LIN {X 0,Y 707.788,Z 622.318,A -85,B 0,C 180,E1 3542.213,E2 3542.213} C_VEL
LIN {X 0,Y 698.542,Z 601.31,A -85,B 0,C 180,E1 3542.971,E2 3542.971} C_VEL
LIN {X 0,Y 698.282,Z 601.31,A -85,B 0,C 180,E1 3548.645,E2 3548.645} C_VEL
LIN {X 0,Y 698.409,Z 601.31,A -85,B 0,C 180,E1 3554.29,E2 3554.29} C_VEL
LIN {X 0,Y 698.252,Z 601.31,A -85,B 0,C 180,E1 3559.425,E2 3559.425} C_VEL
LIN {X 0,Y 698.249,Z 601.31,A -85,B 0,C 180,E1 3564.14,E2 3564.14} C_VEL
LIN {X 0,Y 698.337,Z 601.31,A -85,B 0,C 180,E1 3568.624,E2 3568.624} C_VEL
LIN {X 0,Y 698.426,Z 601.31,A -85,B 0,C 180,E1 3572.902,E2 3572.902} C_VEL
LIN {X 0,Y 698.537,Z 601.31,A -85,B 0,C 180,E1 3577.022,E2 3577.022} C_VEL
LIN {X 0,Y 698.549,Z 601.31,A -85,B 0,C 180,E1 3582.641,E2 3582.641} C_VEL
LIN {X 0,Y 698.415,Z 601.31,A -85,B 0,C 180,E1 3587.509,E2 3587.509} C_VEL
LIN {X 0,Y 698.636,Z 601.31,A -85,B 0,C 180,E1 3592.523,E2 3592.523} C_VEL
LIN {X 0,Y 698.754,Z 601.31,A -85,B 0,C 180,E1 3597.513,E2 3597.513} C_VEL
LIN {X 0,Y 698.624,Z 601.31,A -85,B 0,C 180,E1 3602.484,E2 3602.484} C_VEL
LIN {X 0,Y 698.589,Z 601.31,A -85,B 0,C 180,E1 3606.223,E2 3606.223} C_VEL
LIN {X 0,Y 698.52,Z 601.31,A -85,B 0,C 180,E1 3611.254,E2 3611.254} C_VEL
LIN {X 0,Y 698.581,Z 601.31,A -85,B 0,C 180,E1 3616.372,E2 3616.372} C_VEL
LIN {X 0,Y 698.492,Z 601.31,A -85,B 0,C 180,E1 3621.633,E2 3621.633} C_VEL
LIN {X 0,Y 698.439,Z 601.31,A -85,B 0,C 180,E1 3625.707,E2 3625.707} C_VEL
LIN {X 0,Y 698.346,Z 601.31,A -85,B 0,C 180,E1 3629.927,E2 3629.927} C_VEL
LIN {X 0,Y 698.291,Z 601.31,A -85,B 0,C 180,E1 3634.451,E2 3634.451} C_VEL
LIN {X 0,Y 698.292,Z 601.31,A -85,B 0,C 180,E1 3638.984,E2 3638.984} C_VEL
LIN {X 0,Y 698.437,Z 601.31,A -85,B 0,C 180,E1 3644.277,E2 3644.277} C_VEL
LIN {X 0,Y 698.295,Z 601.31,A -85,B 0,C 180,E1 3649.399,E2 3649.399} C_VEL
LIN {X 0,Y 698.256,Z 601.31,A -85,B 0,C 180,E1 3654.13,E2 3654.13} C_VEL
LIN {X 0,Y 698.361,Z 601.31,A -85,B 0,C 180,E1 3658.616,E2 3658.616} C_VEL
LIN {X 0,Y 698.567,Z 601.31,A -85,B 0,C 180,E1 3664.287,E2 3664.287} C_VEL
LIN {X 0,Y 698.644,Z 601.31,A -85,B 0,C 180,E1 3665.087,E2 3665.087} C_VEL
LIN {X 0,Y 704.33,Z 620.623,A -85,B 0,C 180,E1 3665.608,E2 3665.608} C_VEL
LIN {X 0,Y 703.741,Z 661.307,A -85,B 0,C 180,E1 3666.603,E2 3666.603} C_VEL
LIN {X 0,Y 702.767,Z 699.55,A -85,B 0,C 180,E1 3668.056,E2 3668.056} C_VEL
LIN {X 0,Y 701.625,Z 735.549,A -85,B 0,C 180,E1 3669.988,E2 3669.988} C_VEL
LIN {X 0,Y 700.652,Z 767.288,A -85,B 0,C 180,E1 3672.261,E2 3672.261} C_VEL
LIN {X 0,Y 699.841,Z 795.512,A -85,B 0,C 180,E1 3674.938,E2 3674.938} C_VEL
LIN {X 0,Y 699.357,Z 818.283,A -85,B 0,C 180,E1 3677.801,E2 3677.801} C_VEL
LIN {X 0,Y 699.049,Z 835.787,A -85,B 0,C 180,E1 3680.796,E2 3680.796} C_VEL
LIN {X 0,Y 698.89,Z 847.743,A -85,B 0,C 180,E1 3683.773,E2 3683.773} C_VEL
LIN {X 0,Y 698.874,Z 854.031,A -85,B 0,C 180,E1 3686.267,E2 3686.267} C_VEL
LIN {X 0,Y 698.804,Z 857.085,A -85,B 0,C 180,E1 3688.754,E2 3688.754} C_VEL
LIN {X 0,Y 698.887,Z 857.026,A -85,B 0,C 180,E1 3691.239,E2 3691.239} C_VEL
LIN {X 0,Y 698.999,Z 852.206,A -85,B 0,C 180,E1 3694.519,E2 3694.519} C_VEL
LIN {X 0,Y 699.071,Z 841.77,A -85,B 0,C 180,E1 3697.782,E2 3697.782} C_VEL
LIN {X 0,Y 699.25,Z 825.88,A -85,B 0,C 180,E1 3700.926,E2 3700.926} C_VEL
LIN {X 0,Y 699.701,Z 804.549,A -85,B 0,C 180,E1 3703.937,E2 3703.937} C_VEL
LIN {X 0,Y 700.362,Z 778.69,A -85,B 0,C 180,E1 3706.654,E2 3706.654} C_VEL
LIN {X 0,Y 701.32,Z 747.571,A -85,B 0,C 180,E1 3709.129,E2 3709.129} C_VEL
LIN {X 0,Y 702.354,Z 713.484,A -85,B 0,C 180,E1 3711.18,E2 3711.18} C_VEL
LIN {X 0,Y 703.382,Z 676.025,A -85,B 0,C 180,E1 3712.811,E2 3712.811} C_VEL
LIN {X 0,Y 704.233,Z 635.503,A -85,B 0,C 180,E1 3714,E2 3714} C_VEL
LIN {X 0,Y 703.617,Z 616.54,A -85,B 0,C 180,E1 3714.405,E2 3714.405} C_VEL
LIN {X 0,Y 698.364,Z 601.31,A -85,B 0,C 180,E1 3714.86,E2 3714.86} C_VEL
LIN {X 0,Y 698.363,Z 601.31,A -85,B 0,C 180,E1 3719.931,E2 3719.931} C_VEL
LIN {X 0,Y 698.307,Z 601.31,A -85,B 0,C 180,E1 3724.479,E2 3724.479} C_VEL
LIN {X 0,Y 698.251,Z 601.31,A -85,B 0,C 180,E1 3728.994,E2 3728.994} C_VEL
LIN {X 0,Y 698.44,Z 601.31,A -85,B 0,C 180,E1 3734.297,E2 3734.297} C_VEL
LIN {X 0,Y 698.27,Z 601.31,A -85,B 0,C 180,E1 3739.413,E2 3739.413} C_VEL
LIN {X 0,Y 698.252,Z 601.31,A -85,B 0,C 180,E1 3744.144,E2 3744.144} C_VEL
LIN {X 0,Y 698.338,Z 601.31,A -85,B 0,C 180,E1 3748.628,E2 3748.628} C_VEL
LIN {X 0,Y 698.504,Z 601.31,A -85,B 0,C 180,E1 3754.296,E2 3754.296} C_VEL
LIN {X 0,Y 698.327,Z 601.31,A -85,B 0,C 180,E1 3758.897,E2 3758.897} C_VEL
LIN {X 0,Y 698.394,Z 601.31,A -85,B 0,C 180,E1 3761.57,E2 3761.57} C_VEL
LIN {X 0,Y 702.105,Z 618.347,A -85,B 0,C 180,E1 3761.867,E2 3761.867} C_VEL
LIN {X 0,Y 701.839,Z 691.618,A -85,B 0,C 180,E1 3762.737,E2 3762.737} C_VEL
LIN {X 0,Y 701.426,Z 724.721,A -85,B 0,C 180,E1 3763.615,E2 3763.615} C_VEL
LIN {X 0,Y 700.738,Z 756.316,A -85,B 0,C 180,E1 3764.966,E2 3764.966} C_VEL
LIN {X 0,Y 700.111,Z 785.157,A -85,B 0,C 180,E1 3766.752,E2 3766.752} C_VEL
LIN {X 0,Y 699.572,Z 810.159,A -85,B 0,C 180,E1 3768.921,E2 3768.921} C_VEL
LIN {X 0,Y 699.205,Z 830.58,A -85,B 0,C 180,E1 3771.435,E2 3771.435} C_VEL
LIN {X 0,Y 699.029,Z 845.13,A -85,B 0,C 180,E1 3774.093,E2 3774.093} C_VEL
LIN {X 0,Y 698.976,Z 854.196,A -85,B 0,C 180,E1 3776.896,E2 3776.896} C_VEL
LIN {X 0,Y 698.914,Z 856.955,A -85,B 0,C 180,E1 3778.76,E2 3778.76} C_VEL
LIN {X 0,Y 698.933,Z 856.877,A -85,B 0,C 180,E1 3781.244,E2 3781.244} C_VEL
LIN {X 0,Y 699.024,Z 851.303,A -85,B 0,C 180,E1 3784.126,E2 3784.126} C_VEL
LIN {X 0,Y 699.113,Z 840.282,A -85,B 0,C 180,E1 3786.846,E2 3786.846} C_VEL
LIN {X 0,Y 699.33,Z 823.303,A -85,B 0,C 180,E1 3789.477,E2 3789.477} C_VEL
LIN {X 0,Y 699.742,Z 800.952,A -85,B 0,C 180,E1 3791.87,E2 3791.87} C_VEL
LIN {X 0,Y 700.299,Z 777.418,A -85,B 0,C 180,E1 3793.701,E2 3793.701} C_VEL
LIN {X 0,Y 696.623,Z 764.377,A -85,B 0,C 180,E1 3794.621,E2 3794.621} C_VEL
LIN {X 0,Y 693.254,Z 752.31,A -85,B 0,C 180,E1 3795.348,E2 3795.348} C_VEL
LIN {X 0,Y 693.225,Z 750.405,A -85,B 0,C 180,E1 3795.44,E2 3795.44} C_VEL
LIN {X 0,Y 693.951,Z 717.579,A -85,B 0,C 180,E1 3796.733,E2 3796.733} C_VEL
LIN {X 0,Y 694.411,Z 682.542,A -85,B 0,C 180,E1 3797.539,E2 3797.539} C_VEL
LIN {X 0,Y 694.009,Z 612.919,A -85,B 0,C 180,E1 3798.371,E2 3798.371} C_VEL
LIN {X 0,Y 690.712,Z 601.31,A -85,B 0,C 180,E1 3798.635,E2 3798.635} C_VEL
LIN {X 0,Y 690.49,Z 601.31,A -85,B 0,C 180,E1 3803.262,E2 3803.262} C_VEL
LIN {X 0,Y 690.484,Z 601.31,A -85,B 0,C 180,E1 3808.634,E2 3808.634} C_VEL
LIN {X 0,Y 690.388,Z 601.31,A -85,B 0,C 180,E1 3813.495,E2 3813.495} C_VEL
LIN {X 0,Y 690.456,Z 601.31,A -85,B 0,C 180,E1 3817.905,E2 3817.905} C_VEL
LIN {X 0,Y 690.503,Z 601.31,A -85,B 0,C 180,E1 3823.608,E2 3823.608} C_VEL
LIN {X 0,Y 690.271,Z 601.31,A -85,B 0,C 180,E1 3828.817,E2 3828.817} C_VEL
LIN {X 0,Y 690.311,Z 601.31,A -85,B 0,C 180,E1 3833.66,E2 3833.66} C_VEL
LIN {X 0,Y 690.363,Z 602.018,A -85,B 0,C 180,E1 3836.624,E2 3836.624} C_VEL
LIN {X 0,Y 701.618,Z 627.968,A -85,B 0,C 180,E1 3837.536,E2 3837.536} C_VEL
LIN {X 0,Y 701.063,Z 707.913,A -85,B 0,C 180,E1 3838.565,E2 3838.565} C_VEL
LIN {X 0,Y 700.009,Z 748.6,A -85,B 0,C 180,E1 3839.519,E2 3839.519} C_VEL
LIN {X 0,Y 698.553,Z 792.111,A -85,B 0,C 180,E1 3841.059,E2 3841.059} C_VEL
LIN {X 0,Y 696.858,Z 832.632,A -85,B 0,C 180,E1 3843.039,E2 3843.039} C_VEL
LIN {X 0,Y 695.161,Z 870.148,A -85,B 0,C 180,E1 3845.431,E2 3845.431} C_VEL
LIN {X 0,Y 693.739,Z 904.255,A -85,B 0,C 180,E1 3848.208,E2 3848.208} C_VEL
LIN {X 0,Y 692.563,Z 934.568,A -85,B 0,C 180,E1 3851.343,E2 3851.343} C_VEL
LIN {X 0,Y 691.764,Z 961.239,A -85,B 0,C 180,E1 3854.927,E2 3854.927} C_VEL
LIN {X 0,Y 691.258,Z 981.632,A -85,B 0,C 180,E1 3858.626,E2 3858.626} C_VEL
LIN {X 0,Y 691.102,Z 994.244,A -85,B 0,C 180,E1 3861.81,E2 3861.81} C_VEL
LIN {X 0,Y 690.958,Z 1003.715,A -85,B 0,C 180,E1 3865.625,E2 3865.625} C_VEL
LIN {X 0,Y 691.006,Z 1007.169,A -85,B 0,C 180,E1 3868.747,E2 3868.747} C_VEL
LIN {X 0,Y 691.033,Z 1006.216,A -85,B 0,C 180,E1 3872.517,E2 3872.517} C_VEL
LIN {X 0,Y 690.976,Z 999.627,A -85,B 0,C 180,E1 3876.298,E2 3876.298} C_VEL
LIN {X 0,Y 691.137,Z 988.788,A -85,B 0,C 180,E1 3879.717,E2 3879.717} C_VEL
LIN {X 0,Y 691.37,Z 970.858,A -85,B 0,C 180,E1 3883.475,E2 3883.475} C_VEL
LIN {X 0,Y 691.911,Z 949.955,A -85,B 0,C 180,E1 3886.707,E2 3886.707} C_VEL
LIN {X 0,Y 692.876,Z 923.253,A -85,B 0,C 180,E1 3889.921,E2 3889.921} C_VEL
LIN {X 0,Y 694.331,Z 889.898,A -85,B 0,C 180,E1 3893.048,E2 3893.048} C_VEL
LIN {X 0,Y 696.009,Z 851.914,A -85,B 0,C 180,E1 3895.814,E2 3895.814} C_VEL
LIN {X 0,Y 697.776,Z 811.008,A -85,B 0,C 180,E1 3898.09,E2 3898.09} C_VEL
LIN {X 0,Y 699.268,Z 772.005,A -85,B 0,C 180,E1 3899.718,E2 3899.718} C_VEL
LIN {X 0,Y 700.658,Z 729.711,A -85,B 0,C 180,E1 3900.979,E2 3900.979} C_VEL
LIN {X 0,Y 701.336,Z 686.179,A -85,B 0,C 180,E1 3901.776,E2 3901.776} C_VEL
LIN {X 0,Y 701.268,Z 625.08,A -85,B 0,C 180,E1 3902.516,E2 3902.516} C_VEL
LIN {X 0,Y 690.525,Z 601.31,A -85,B 0,C 180,E1 3903.414,E2 3903.414} C_VEL
LIN {X 0,Y 690.391,Z 601.31,A -85,B 0,C 180,E1 3907.921,E2 3907.921} C_VEL
LIN {X 0,Y 690.469,Z 601.31,A -85,B 0,C 180,E1 3913.611,E2 3913.611} C_VEL
LIN {X 0,Y 690.275,Z 601.31,A -85,B 0,C 180,E1 3918.821,E2 3918.821} C_VEL
LIN {X 0,Y 690.342,Z 601.31,A -85,B 0,C 180,E1 3923.664,E2 3923.664} C_VEL
LIN {X 0,Y 690.429,Z 601.31,A -85,B 0,C 180,E1 3928.865,E2 3928.865} C_VEL
LIN {X 0,Y 690.568,Z 601.31,A -85,B 0,C 180,E1 3934.113,E2 3934.113} C_VEL
LIN {X 0,Y 690.562,Z 601.31,A -85,B 0,C 180,E1 3938.102,E2 3938.102} C_VEL
LIN {X 0,Y 690.617,Z 601.31,A -85,B 0,C 180,E1 3943.43,E2 3943.43} C_VEL
LIN {X 0,Y 690.638,Z 601.31,A -85,B 0,C 180,E1 3948.613,E2 3948.613} C_VEL
LIN {X 0,Y 690.785,Z 601.31,A -85,B 0,C 180,E1 3953.703,E2 3953.703} C_VEL
LIN {X 0,Y 690.738,Z 601.31,A -85,B 0,C 180,E1 3958.742,E2 3958.742} C_VEL
LIN {X 0,Y 690.741,Z 601.31,A -85,B 0,C 180,E1 3962.512,E2 3962.512} C_VEL
LIN {X 0,Y 690.68,Z 601.31,A -85,B 0,C 180,E1 3966.294,E2 3966.294} C_VEL
LIN {X 0,Y 690.644,Z 601.31,A -85,B 0,C 180,E1 3971.384,E2 3971.384} C_VEL
LIN {X 0,Y 690.683,Z 601.31,A -85,B 0,C 180,E1 3976.565,E2 3976.565} C_VEL
LIN {X 0,Y 690.558,Z 601.31,A -85,B 0,C 180,E1 3981.895,E2 3981.895} C_VEL
LIN {X 0,Y 690.505,Z 601.31,A -85,B 0,C 180,E1 3986.024,E2 3986.024} C_VEL
LIN {X 0,Y 690.432,Z 601.31,A -85,B 0,C 180,E1 3991.136,E2 3991.136} C_VEL
LIN {X 0,Y 690.429,Z 601.31,A -85,B 0,C 180,E1 3996.326,E2 3996.326} C_VEL
LIN {X 0,Y 690.409,Z 601.31,A -85,B 0,C 180,E1 4001.734,E2 4001.734} C_VEL
LIN {X 0,Y 690.35,Z 601.31,A -85,B 0,C 180,E1 4006.395,E2 4006.395} C_VEL
LIN {X 0,Y 690.377,Z 601.31,A -85,B 0,C 180,E1 4012.177,E2 4012.177} C_VEL
LIN {X 0,Y 690.34,Z 601.31,A -85,B 0,C 180,E1 4016.717,E2 4016.717} C_VEL
LIN {X 0,Y 690.493,Z 601.31,A -85,B 0,C 180,E1 4021.347,E2 4021.347} C_VEL
LIN {X 0,Y 690.725,Z 601.31,A -85,B 0,C 180,E1 4024.781,E2 4024.781} C_VEL
LIN {X 0,Y 697.118,Z 622.821,A -85,B 0,C 180,E1 4025.383,E2 4025.383} C_VEL
LIN {X 0,Y 696.426,Z 663.052,A -85,B 0,C 180,E1 4026.397,E2 4026.397} C_VEL
LIN {X 0,Y 695.307,Z 700.604,A -85,B 0,C 180,E1 4027.861,E2 4027.861} C_VEL
LIN {X 0,Y 694.055,Z 736.725,A -85,B 0,C 180,E1 4029.836,E2 4029.836} C_VEL
LIN {X 0,Y 692.938,Z 768.609,A -85,B 0,C 180,E1 4032.17,E2 4032.17} C_VEL
LIN {X 0,Y 692.103,Z 795.501,A -85,B 0,C 180,E1 4034.765,E2 4034.765} C_VEL
LIN {X 0,Y 691.527,Z 818.279,A -85,B 0,C 180,E1 4037.661,E2 4037.661} C_VEL
LIN {X 0,Y 691.197,Z 834.771,A -85,B 0,C 180,E1 4040.48,E2 4040.48} C_VEL
LIN {X 0,Y 690.996,Z 847.743,A -85,B 0,C 180,E1 4043.702,E2 4043.702} C_VEL
LIN {X 0,Y 690.984,Z 854.033,A -85,B 0,C 180,E1 4046.225,E2 4046.225} C_VEL
LIN {X 0,Y 690.911,Z 857.08,A -85,B 0,C 180,E1 4048.74,E2 4048.74} C_VEL
LIN {X 0,Y 690.989,Z 857.021,A -85,B 0,C 180,E1 4051.253,E2 4051.253} C_VEL
LIN {X 0,Y 691.099,Z 852.201,A -85,B 0,C 180,E1 4054.571,E2 4054.571} C_VEL
LIN {X 0,Y 691.166,Z 841.774,A -85,B 0,C 180,E1 4057.872,E2 4057.872} C_VEL
LIN {X 0,Y 691.426,Z 825.878,A -85,B 0,C 180,E1 4061.051,E2 4061.051} C_VEL
LIN {X 0,Y 691.895,Z 804.554,A -85,B 0,C 180,E1 4064.097,E2 4064.097} C_VEL
LIN {X 0,Y 692.653,Z 778.7,A -85,B 0,C 180,E1 4066.845,E2 4066.845} C_VEL
LIN {X 0,Y 693.687,Z 748.784,A -85,B 0,C 180,E1 4069.261,E2 4069.261} C_VEL
LIN {X 0,Y 694.853,Z 715.017,A -85,B 0,C 180,E1 4071.336,E2 4071.336} C_VEL
LIN {X 0,Y 695.978,Z 678.621,A -85,B 0,C 180,E1 4072.972,E2 4072.972} C_VEL
LIN {X 0,Y 696.933,Z 637.993,A -85,B 0,C 180,E1 4074.205,E2 4074.205} C_VEL
LIN {X 0,Y 696.408,Z 618.768,A -85,B 0,C 180,E1 4074.632,E2 4074.632} C_VEL
LIN {X 0,Y 690.439,Z 601.31,A -85,B 0,C 180,E1 4075.145,E2 4075.145} C_VEL
LIN {X 0,Y 690.421,Z 601.31,A -85,B 0,C 180,E1 4080.311,E2 4080.311} C_VEL
LIN {X 0,Y 690.396,Z 601.31,A -85,B 0,C 180,E1 4085.725,E2 4085.725} C_VEL
LIN {X 0,Y 690.327,Z 601.31,A -85,B 0,C 180,E1 4091.179,E2 4091.179} C_VEL
LIN {X 0,Y 690.433,Z 601.31,A -85,B 0,C 180,E1 4095.405,E2 4095.405} C_VEL
LIN {X 0,Y 690.317,Z 601.31,A -85,B 0,C 180,E1 4100.478,E2 4100.478} C_VEL
LIN {X 0,Y 690.325,Z 601.31,A -85,B 0,C 180,E1 4105.213,E2 4105.213} C_VEL
LIN {X 0,Y 690.402,Z 601.31,A -85,B 0,C 180,E1 4109.693,E2 4109.693} C_VEL
LIN {X 0,Y 690.587,Z 601.31,A -85,B 0,C 180,E1 4114.094,E2 4114.094} C_VEL
LIN {X 0,Y 690.488,Z 601.31,A -85,B 0,C 180,E1 4118.103,E2 4118.103} C_VEL
LIN {X 0,Y 690.45,Z 601.31,A -85,B 0,C 180,E1 4121.341,E2 4121.341} C_VEL
LIN {X 0,Y 694.653,Z 618.658,A -85,B 0,C 180,E1 4121.655,E2 4121.655} C_VEL
LIN {X 0,Y 694.336,Z 690.008,A -85,B 0,C 180,E1 4122.504,E2 4122.504} C_VEL
LIN {X 0,Y 693.867,Z 723.802,A -85,B 0,C 180,E1 4123.391,E2 4123.391} C_VEL
LIN {X 0,Y 693.115,Z 754.803,A -85,B 0,C 180,E1 4124.699,E2 4124.699} C_VEL
LIN {X 0,Y 692.445,Z 783.749,A -85,B 0,C 180,E1 4126.482,E2 4126.482} C_VEL
LIN {X 0,Y 691.778,Z 808.559,A -85,B 0,C 180,E1 4128.635,E2 4128.635} C_VEL
LIN {X 0,Y 691.41,Z 828.174,A -85,B 0,C 180,E1 4130.987,E2 4130.987} C_VEL
LIN {X 0,Y 691.181,Z 843.788,A -85,B 0,C 180,E1 4133.71,E2 4133.71} C_VEL
LIN {X 0,Y 691.113,Z 852.678,A -85,B 0,C 180,E1 4136.231,E2 4136.231} C_VEL
LIN {X 0,Y 691.021,Z 856.954,A -85,B 0,C 180,E1 4138.745,E2 4138.745} C_VEL
LIN {X 0,Y 691.038,Z 856.877,A -85,B 0,C 180,E1 4141.258,E2 4141.258} C_VEL
LIN {X 0,Y 691.125,Z 851.49,A -85,B 0,C 180,E1 4144.112,E2 4144.112} C_VEL
LIN {X 0,Y 691.229,Z 840.285,A -85,B 0,C 180,E1 4146.925,E2 4146.925} C_VEL
LIN {X 0,Y 691.469,Z 823.248,A -85,B 0,C 180,E1 4149.593,E2 4149.593} C_VEL
LIN {X 0,Y 691.942,Z 800.972,A -85,B 0,C 180,E1 4152.006,E2 4152.006} C_VEL
LIN {X 0,Y 692.635,Z 775.636,A -85,B 0,C 180,E1 4154.003,E2 4154.003} C_VEL
LIN {X 0,Y 693.225,Z 750.405,A -85,B 0,C 180,E1 4155.44,E2 4155.44} C_VEL
LIN {X 0,Y 689.935,Z 735.712,A -85,B 0,C 180,E1 4156.19,E2 4156.19} C_VEL
LIN {X 0,Y 686.319,Z 721.512,A -85,B 0,C 180,E1 4156.808,E2 4156.808} C_VEL
LIN {X 0,Y 686.329,Z 720.499,A -85,B 0,C 180,E1 4156.843,E2 4156.843} C_VEL
LIN {X 0,Y 686.892,Z 685.627,A -85,B 0,C 180,E1 4157.696,E2 4157.696} C_VEL
LIN {X 0,Y 686.499,Z 613.882,A -85,B 0,C 180,E1 4158.596,E2 4158.596} C_VEL
LIN {X 0,Y 682.779,Z 601.31,A -85,B 0,C 180,E1 4158.92,E2 4158.92} C_VEL
LIN {X 0,Y 682.567,Z 601.31,A -85,B 0,C 180,E1 4164.483,E2 4164.483} C_VEL
LIN {X 0,Y 682.51,Z 601.31,A -85,B 0,C 180,E1 4169.231,E2 4169.231} C_VEL
LIN {X 0,Y 682.523,Z 601.31,A -85,B 0,C 180,E1 4174.781,E2 4174.781} C_VEL
LIN {X 0,Y 682.402,Z 601.31,A -85,B 0,C 180,E1 4180.076,E2 4180.076} C_VEL
LIN {X 0,Y 682.593,Z 601.31,A -85,B 0,C 180,E1 4184.743,E2 4184.743} C_VEL
LIN {X 0,Y 682.366,Z 601.31,A -85,B 0,C 180,E1 4189.918,E2 4189.918} C_VEL
LIN {X 0,Y 682.375,Z 601.31,A -85,B 0,C 180,E1 4195.228,E2 4195.228} C_VEL
LIN {X 0,Y 682.39,Z 601.31,A -85,B 0,C 180,E1 4196.166,E2 4196.166} C_VEL
LIN {X 0,Y 694.974,Z 629.987,A -85,B 0,C 180,E1 4197.212,E2 4197.212} C_VEL
LIN {X 0,Y 694.299,Z 708.221,A -85,B 0,C 180,E1 4198.229,E2 4198.229} C_VEL
LIN {X 0,Y 693.162,Z 748.575,A -85,B 0,C 180,E1 4199.185,E2 4199.185} C_VEL
LIN {X 0,Y 691.58,Z 791.241,A -85,B 0,C 180,E1 4200.702,E2 4200.702} C_VEL
LIN {X 0,Y 689.771,Z 830.846,A -85,B 0,C 180,E1 4202.636,E2 4202.636} C_VEL
LIN {X 0,Y 687.947,Z 867.704,A -85,B 0,C 180,E1 4204.972,E2 4204.972} C_VEL
LIN {X 0,Y 686.216,Z 902.493,A -85,B 0,C 180,E1 4207.786,E2 4207.786} C_VEL
LIN {X 0,Y 684.879,Z 934.568,A -85,B 0,C 180,E1 4211.125,E2 4211.125} C_VEL
LIN {X 0,Y 683.955,Z 961.237,A -85,B 0,C 180,E1 4214.751,E2 4214.751} C_VEL
LIN {X 0,Y 683.396,Z 981.631,A -85,B 0,C 180,E1 4218.493,E2 4218.493} C_VEL
LIN {X 0,Y 683.232,Z 994.244,A -85,B 0,C 180,E1 4221.715,E2 4221.715} C_VEL
LIN {X 0,Y 683.077,Z 1003.671,A -85,B 0,C 180,E1 4225.551,E2 4225.551} C_VEL
LIN {X 0,Y 683.103,Z 1007.169,A -85,B 0,C 180,E1 4228.733,E2 4228.733} C_VEL
LIN {X 0,Y 683.127,Z 1006.215,A -85,B 0,C 180,E1 4232.546,E2 4232.546} C_VEL
LIN {X 0,Y 683.155,Z 1001.188,A -85,B 0,C 180,E1 4235.732,E2 4235.732} C_VEL
LIN {X 0,Y 683.235,Z 989.724,A -85,B 0,C 180,E1 4239.572,E2 4239.572} C_VEL
LIN {X 0,Y 683.523,Z 973.523,A -85,B 0,C 180,E1 4243.137,E2 4243.137} C_VEL
LIN {X 0,Y 684.066,Z 952.358,A -85,B 0,C 180,E1 4246.573,E2 4246.573} C_VEL
LIN {X 0,Y 685.197,Z 924.381,A -85,B 0,C 180,E1 4250.034,E2 4250.034} C_VEL
LIN {X 0,Y 686.821,Z 889.899,A -85,B 0,C 180,E1 4253.315,E2 4253.315} C_VEL
LIN {X 0,Y 688.737,Z 851.914,A -85,B 0,C 180,E1 4256.107,E2 4256.107} C_VEL
LIN {X 0,Y 690.658,Z 810.743,A -85,B 0,C 180,E1 4258.419,E2 4258.419} C_VEL
LIN {X 0,Y 692.377,Z 770.375,A -85,B 0,C 180,E1 4260.105,E2 4260.105} C_VEL
LIN {X 0,Y 693.839,Z 729.451,A -85,B 0,C 180,E1 4261.324,E2 4261.324} C_VEL
LIN {X 0,Y 694.646,Z 685.297,A -85,B 0,C 180,E1 4262.131,E2 4262.131} C_VEL
LIN {X 0,Y 694.462,Z 627.246,A -85,B 0,C 180,E1 4262.849,E2 4262.849} C_VEL
LIN {X 0,Y 682.565,Z 601.31,A -85,B 0,C 180,E1 4263.847,E2 4263.847} C_VEL
LIN {X 0,Y 682.38,Z 601.31,A -85,B 0,C 180,E1 4269.011,E2 4269.011} C_VEL
LIN {X 0,Y 682.563,Z 601.31,A -85,B 0,C 180,E1 4273.49,E2 4273.49} C_VEL
LIN {X 0,Y 682.376,Z 601.31,A -85,B 0,C 180,E1 4279.028,E2 4279.028} C_VEL
LIN {X 0,Y 682.394,Z 601.31,A -85,B 0,C 180,E1 4283.172,E2 4283.172} C_VEL
LIN {X 0,Y 682.435,Z 601.31,A -85,B 0,C 180,E1 4287.806,E2 4287.806} C_VEL
LIN {X 0,Y 682.624,Z 601.31,A -85,B 0,C 180,E1 4292.614,E2 4292.614} C_VEL
LIN {X 0,Y 682.664,Z 601.31,A -85,B 0,C 180,E1 4297.835,E2 4297.835} C_VEL
LIN {X 0,Y 682.692,Z 601.31,A -85,B 0,C 180,E1 4303.232,E2 4303.232} C_VEL
LIN {X 0,Y 682.708,Z 601.31,A -85,B 0,C 180,E1 4308.479,E2 4308.479} C_VEL
LIN {X 0,Y 682.901,Z 601.31,A -85,B 0,C 180,E1 4313.63,E2 4313.63} C_VEL
LIN {X 0,Y 682.839,Z 601.31,A -85,B 0,C 180,E1 4318.727,E2 4318.727} C_VEL
LIN {X 0,Y 682.862,Z 601.31,A -85,B 0,C 180,E1 4323.068,E2 4323.068} C_VEL
LIN {X 0,Y 682.782,Z 601.31,A -85,B 0,C 180,E1 4327.648,E2 4327.648} C_VEL
LIN {X 0,Y 682.778,Z 601.31,A -85,B 0,C 180,E1 4332.817,E2 4332.817} C_VEL
LIN {X 0,Y 682.708,Z 601.31,A -85,B 0,C 180,E1 4338.097,E2 4338.097} C_VEL
LIN {X 0,Y 682.613,Z 601.31,A -85,B 0,C 180,E1 4343.543,E2 4343.543} C_VEL
LIN {X 0,Y 682.576,Z 601.31,A -85,B 0,C 180,E1 4347.777,E2 4347.777} C_VEL
LIN {X 0,Y 682.459,Z 601.31,A -85,B 0,C 180,E1 4352.463,E2 4352.463} C_VEL
LIN {X 0,Y 682.483,Z 601.31,A -85,B 0,C 180,E1 4356.936,E2 4356.936} C_VEL
LIN {X 0,Y 682.589,Z 601.31,A -85,B 0,C 180,E1 4362.896,E2 4362.896} C_VEL
LIN {X 0,Y 682.407,Z 601.31,A -85,B 0,C 180,E1 4368.227,E2 4368.227} C_VEL
LIN {X 0,Y 682.408,Z 601.31,A -85,B 0,C 180,E1 4373.161,E2 4373.161} C_VEL
LIN {X 0,Y 682.467,Z 601.31,A -85,B 0,C 180,E1 4377.798,E2 4377.798} C_VEL
LIN {X 0,Y 682.663,Z 601.31,A -85,B 0,C 180,E1 4382.574,E2 4382.574} C_VEL
LIN {X 0,Y 682.799,Z 601.31,A -85,B 0,C 180,E1 4384.457,E2 4384.457} C_VEL
LIN {X 0,Y 689.909,Z 624.36,A -85,B 0,C 180,E1 4385.14,E2 4385.14} C_VEL
LIN {X 0,Y 689.131,Z 663.874,A -85,B 0,C 180,E1 4386.158,E2 4386.158} C_VEL
LIN {X 0,Y 687.857,Z 701.615,A -85,B 0,C 180,E1 4387.66,E2 4387.66} C_VEL
LIN {X 0,Y 686.463,Z 738.394,A -85,B 0,C 180,E1 4389.713,E2 4389.713} C_VEL
LIN {X 0,Y 685.205,Z 770.515,A -85,B 0,C 180,E1 4392.129,E2 4392.129} C_VEL
LIN {X 0,Y 684.235,Z 798.363,A -85,B 0,C 180,E1 4394.915,E2 4394.915} C_VEL
LIN {X 0,Y 683.661,Z 821.506,A -85,B 0,C 180,E1 4398.004,E2 4398.004} C_VEL
LIN {X 0,Y 683.26,Z 838.009,A -85,B 0,C 180,E1 4401.066,E2 4401.066} C_VEL
LIN {X 0,Y 683.161,Z 849.602,A -85,B 0,C 180,E1 4404.268,E2 4404.268} C_VEL
LIN {X 0,Y 683.114,Z 855.945,A -85,B 0,C 180,E1 4407.454,E2 4407.454} C_VEL
LIN {X 0,Y 683.008,Z 857.439,A -85,B 0,C 180,E1 4409.996,E2 4409.996} C_VEL
LIN {X 0,Y 683.084,Z 855.835,A -85,B 0,C 180,E1 4412.539,E2 4412.539} C_VEL
LIN {X 0,Y 683.172,Z 849.365,A -85,B 0,C 180,E1 4415.724,E2 4415.724} C_VEL
LIN {X 0,Y 683.259,Z 837.647,A -85,B 0,C 180,E1 4418.927,E2 4418.927} C_VEL
LIN {X 0,Y 683.671,Z 819.906,A -85,B 0,C 180,E1 4422.151,E2 4422.151} C_VEL
LIN {X 0,Y 684.22,Z 797.639,A -85,B 0,C 180,E1 4425.079,E2 4425.079} C_VEL
LIN {X 0,Y 685.277,Z 769.573,A -85,B 0,C 180,E1 4427.862,E2 4427.862} C_VEL
LIN {X 0,Y 686.458,Z 738.588,A -85,B 0,C 180,E1 4430.185,E2 4430.185} C_VEL
LIN {X 0,Y 687.81,Z 702.523,A -85,B 0,C 180,E1 4432.206,E2 4432.206} C_VEL
LIN {X 0,Y 689.096,Z 665.763,A -85,B 0,C 180,E1 4433.69,E2 4433.69} C_VEL
LIN {X 0,Y 689.952,Z 627.802,A -85,B 0,C 180,E1 4434.701,E2 4434.701} C_VEL
LIN {X 0,Y 688.662,Z 619.153,A -85,B 0,C 180,E1 4434.92,E2 4434.92} C_VEL
LIN {X 0,Y 682.507,Z 601.31,A -85,B 0,C 180,E1 4435.507,E2 4435.507} C_VEL
LIN {X 0,Y 682.543,Z 601.31,A -85,B 0,C 180,E1 4440.699,E2 4440.699} C_VEL
LIN {X 0,Y 682.488,Z 601.31,A -85,B 0,C 180,E1 4445.252,E2 4445.252} C_VEL
LIN {X 0,Y 682.375,Z 601.31,A -85,B 0,C 180,E1 4450.082,E2 4450.082} C_VEL
LIN {X 0,Y 682.582,Z 601.31,A -85,B 0,C 180,E1 4454.752,E2 4454.752} C_VEL
LIN {X 0,Y 682.386,Z 601.31,A -85,B 0,C 180,E1 4459.927,E2 4459.927} C_VEL
LIN {X 0,Y 682.451,Z 601.31,A -85,B 0,C 180,E1 4465.228,E2 4465.228} C_VEL
LIN {X 0,Y 682.481,Z 601.31,A -85,B 0,C 180,E1 4470.771,E2 4470.771} C_VEL
LIN {X 0,Y 682.682,Z 601.31,A -85,B 0,C 180,E1 4475.495,E2 4475.495} C_VEL
LIN {X 0,Y 682.514,Z 601.31,A -85,B 0,C 180,E1 4481.091,E2 4481.091} C_VEL
LIN {X 0,Y 687.194,Z 620.641,A -85,B 0,C 180,E1 4481.457,E2 4481.457} C_VEL
LIN {X 0,Y 686.785,Z 692.319,A -85,B 0,C 180,E1 4482.346,E2 4482.346} C_VEL
LIN {X 0,Y 686.26,Z 726.514,A -85,B 0,C 180,E1 4483.284,E2 4483.284} C_VEL
LIN {X 0,Y 685.473,Z 757.013,A -85,B 0,C 180,E1 4484.623,E2 4484.623} C_VEL
LIN {X 0,Y 684.673,Z 786.281,A -85,B 0,C 180,E1 4486.484,E2 4486.484} C_VEL
LIN {X 0,Y 683.984,Z 810.594,A -85,B 0,C 180,E1 4488.666,E2 4488.666} C_VEL
LIN {X 0,Y 683.523,Z 829.634,A -85,B 0,C 180,E1 4491.077,E2 4491.077} C_VEL
LIN {X 0,Y 683.298,Z 845.126,A -85,B 0,C 180,E1 4493.957,E2 4493.957} C_VEL
LIN {X 0,Y 683.2,Z 853.909,A -85,B 0,C 180,E1 4496.69,E2 4496.69} C_VEL
LIN {X 0,Y 683.12,Z 856.953,A -85,B 0,C 180,E1 4498.731,E2 4498.731} C_VEL
LIN {X 0,Y 683.137,Z 856.877,A -85,B 0,C 180,E1 4501.272,E2 4501.272} C_VEL
LIN {X 0,Y 683.231,Z 852.447,A -85,B 0,C 180,E1 4503.816,E2 4503.816} C_VEL
LIN {X 0,Y 683.343,Z 841.82,A -85,B 0,C 180,E1 4506.685,E2 4506.685} C_VEL
LIN {X 0,Y 683.626,Z 825.894,A -85,B 0,C 180,E1 4509.396,E2 4509.396} C_VEL
LIN {X 0,Y 684.15,Z 805.221,A -85,B 0,C 180,E1 4511.821,E2 4511.821} C_VEL
LIN {X 0,Y 684.927,Z 779.51,A -85,B 0,C 180,E1 4513.941,E2 4513.941} C_VEL
LIN {X 0,Y 685.626,Z 750.985,A -85,B 0,C 180,E1 4515.615,E2 4515.615} C_VEL
LIN {X 0,Y 686.329,Z 720.499,A -85,B 0,C 180,E1 4516.843,E2 4516.843} C_VEL
LIN {X 0,Y 682.795,Z 704.662,A -85,B 0,C 180,E1 4517.414,E2 4517.414} C_VEL
LIN {X 0,Y 679.342,Z 690.511,A -85,B 0,C 180,E1 4517.823,E2 4517.823} C_VEL
LIN {X 0,Y 679.322,Z 688.373,A -85,B 0,C 180,E1 4517.862,E2 4517.862} C_VEL
LIN {X 0,Y 679.131,Z 615.453,A -85,B 0,C 180,E1 4518.814,E2 4518.814} C_VEL
LIN {X 0,Y 674.84,Z 601.31,A -85,B 0,C 180,E1 4519.18,E2 4519.18} C_VEL
LIN {X 0,Y 674.642,Z 601.31,A -85,B 0,C 180,E1 4523.842,E2 4523.842} C_VEL
LIN {X 0,Y 674.583,Z 601.31,A -85,B 0,C 180,E1 4528.845,E2 4528.845} C_VEL
LIN {X 0,Y 674.603,Z 601.31,A -85,B 0,C 180,E1 4534.154,E2 4534.154} C_VEL
LIN {X 0,Y 674.539,Z 601.31,A -85,B 0,C 180,E1 4538.966,E2 4538.966} C_VEL
LIN {X 0,Y 674.662,Z 601.31,A -85,B 0,C 180,E1 4544.115,E2 4544.115} C_VEL
LIN {X 0,Y 674.478,Z 601.31,A -85,B 0,C 180,E1 4549.789,E2 4549.789} C_VEL
LIN {X 0,Y 674.485,Z 601.31,A -85,B 0,C 180,E1 4555.355,E2 4555.355} C_VEL
LIN {X 0,Y 674.48,Z 601.31,A -85,B 0,C 180,E1 4555.749,E2 4555.749} C_VEL
LIN {X 0,Y 686.405,Z 627.673,A -85,B 0,C 180,E1 4556.721,E2 4556.721} C_VEL
LIN {X 0,Y 688.361,Z 633.14,A -85,B 0,C 180,E1 4556.895,E2 4556.895} C_VEL
LIN {X 0,Y 687.584,Z 708.394,A -85,B 0,C 180,E1 4557.885,E2 4557.885} C_VEL
LIN {X 0,Y 686.278,Z 749.265,A -85,B 0,C 180,E1 4558.864,E2 4558.864} C_VEL
LIN {X 0,Y 684.534,Z 792.897,A -85,B 0,C 180,E1 4560.441,E2 4560.441} C_VEL
LIN {X 0,Y 682.477,Z 832.966,A -85,B 0,C 180,E1 4562.443,E2 4562.443} C_VEL
LIN {X 0,Y 680.483,Z 869.502,A -85,B 0,C 180,E1 4564.816,E2 4564.816} C_VEL
LIN {X 0,Y 678.598,Z 904.256,A -85,B 0,C 180,E1 4567.696,E2 4567.696} C_VEL
LIN {X 0,Y 677.18,Z 934.568,A -85,B 0,C 180,E1 4570.903,E2 4570.903} C_VEL
LIN {X 0,Y 676.129,Z 961.21,A -85,B 0,C 180,E1 4574.566,E2 4574.566} C_VEL
LIN {X 0,Y 675.547,Z 981.63,A -85,B 0,C 180,E1 4578.358,E2 4578.358} C_VEL
LIN {X 0,Y 675.351,Z 994.244,A -85,B 0,C 180,E1 4581.618,E2 4581.618} C_VEL
LIN {X 0,Y 675.18,Z 1003.671,A -85,B 0,C 180,E1 4585.499,E2 4585.499} C_VEL
LIN {X 0,Y 675.231,Z 1007.169,A -85,B 0,C 180,E1 4588.718,E2 4588.718} C_VEL
LIN {X 0,Y 675.225,Z 1006.215,A -85,B 0,C 180,E1 4592.576,E2 4592.576} C_VEL
LIN {X 0,Y 675.275,Z 1001.188,A -85,B 0,C 180,E1 4595.799,E2 4595.799} C_VEL
LIN {X 0,Y 675.343,Z 989.577,A -85,B 0,C 180,E1 4599.727,E2 4599.727} C_VEL
LIN {X 0,Y 675.664,Z 973.522,A -85,B 0,C 180,E1 4603.292,E2 4603.292} C_VEL
LIN {X 0,Y 676.293,Z 952.356,A -85,B 0,C 180,E1 4606.769,E2 4606.769} C_VEL
LIN {X 0,Y 677.548,Z 924.908,A -85,B 0,C 180,E1 4610.209,E2 4610.209} C_VEL
LIN {X 0,Y 679.29,Z 890.911,A -85,B 0,C 180,E1 4613.502,E2 4613.502} C_VEL
LIN {X 0,Y 681.484,Z 851.913,A -85,B 0,C 180,E1 4616.407,E2 4616.407} C_VEL
LIN {X 0,Y 683.582,Z 811.188,A -85,B 0,C 180,E1 4618.716,E2 4618.716} C_VEL
LIN {X 0,Y 685.455,Z 770.662,A -85,B 0,C 180,E1 4620.43,E2 4620.43} C_VEL
LIN {X 0,Y 687.032,Z 730.129,A -85,B 0,C 180,E1 4621.652,E2 4621.652} C_VEL
LIN {X 0,Y 687.931,Z 687.835,A -85,B 0,C 180,E1 4622.446,E2 4622.446} C_VEL
LIN {X 0,Y 687.791,Z 629.854,A -85,B 0,C 180,E1 4623.176,E2 4623.176} C_VEL
LIN {X 0,Y 674.622,Z 601.31,A -85,B 0,C 180,E1 4624.287,E2 4624.287} C_VEL
LIN {X 0,Y 674.502,Z 601.31,A -85,B 0,C 180,E1 4628.98,E2 4628.98} C_VEL
LIN {X 0,Y 674.622,Z 601.31,A -85,B 0,C 180,E1 4634.133,E2 4634.133} C_VEL
LIN {X 0,Y 674.5,Z 601.31,A -85,B 0,C 180,E1 4639.804,E2 4639.804} C_VEL
LIN {X 0,Y 674.449,Z 601.31,A -85,B 0,C 180,E1 4644.267,E2 4644.267} C_VEL
LIN {X 0,Y 674.535,Z 601.31,A -85,B 0,C 180,E1 4648.898,E2 4648.898} C_VEL
LIN {X 0,Y 674.681,Z 601.31,A -85,B 0,C 180,E1 4653.947,E2 4653.947} C_VEL
LIN {X 0,Y 674.733,Z 601.31,A -85,B 0,C 180,E1 4658.946,E2 4658.946} C_VEL
LIN {X 0,Y 674.782,Z 601.31,A -85,B 0,C 180,E1 4664.37,E2 4664.37} C_VEL
LIN {X 0,Y 674.865,Z 601.31,A -85,B 0,C 180,E1 4669.653,E2 4669.653} C_VEL
LIN {X 0,Y 674.903,Z 601.31,A -85,B 0,C 180,E1 4674.847,E2 4674.847} C_VEL
LIN {X 0,Y 675.008,Z 601.31,A -85,B 0,C 180,E1 4679.998,E2 4679.998} C_VEL
LIN {X 0,Y 675.109,Z 601.31,A -85,B 0,C 180,E1 4685.148,E2 4685.148} C_VEL
LIN {X 0,Y 674.828,Z 601.31,A -85,B 0,C 180,E1 4690.344,E2 4690.344} C_VEL
LIN {X 0,Y 674.805,Z 601.31,A -85,B 0,C 180,E1 4695.626,E2 4695.626} C_VEL
LIN {X 0,Y 674.766,Z 601.31,A -85,B 0,C 180,E1 4701.05,E2 4701.05} C_VEL
LIN {X 0,Y 674.659,Z 601.31,A -85,B 0,C 180,E1 4706.683,E2 4706.683} C_VEL
LIN {X 0,Y 674.549,Z 601.31,A -85,B 0,C 180,E1 4711.391,E2 4711.391} C_VEL
LIN {X 0,Y 674.522,Z 601.31,A -85,B 0,C 180,E1 4716.027,E2 4716.027} C_VEL
LIN {X 0,Y 674.522,Z 601.31,A -85,B 0,C 180,E1 4720.637,E2 4720.637} C_VEL
LIN {X 0,Y 674.575,Z 601.31,A -85,B 0,C 180,E1 4725.938,E2 4725.938} C_VEL
LIN {X 0,Y 674.51,Z 601.31,A -85,B 0,C 180,E1 4731.02,E2 4731.02} C_VEL
LIN {X 0,Y 674.529,Z 601.31,A -85,B 0,C 180,E1 4736.195,E2 4736.195} C_VEL
LIN {X 0,Y 674.586,Z 601.31,A -85,B 0,C 180,E1 4741.137,E2 4741.137} C_VEL
LIN {X 0,Y 674.866,Z 601.31,A -85,B 0,C 180,E1 4744.156,E2 4744.156} C_VEL
LIN {X 0,Y 682.737,Z 626.862,A -85,B 0,C 180,E1 4744.912,E2 4744.912} C_VEL
LIN {X 0,Y 681.819,Z 665.353,A -85,B 0,C 180,E1 4745.936,E2 4745.936} C_VEL
LIN {X 0,Y 680.42,Z 703.172,A -85,B 0,C 180,E1 4747.483,E2 4747.483} C_VEL
LIN {X 0,Y 678.941,Z 738.895,A -85,B 0,C 180,E1 4749.512,E2 4749.512} C_VEL
LIN {X 0,Y 677.539,Z 770.741,A -85,B 0,C 180,E1 4751.942,E2 4751.942} C_VEL
LIN {X 0,Y 676.484,Z 798.351,A -85,B 0,C 180,E1 4754.738,E2 4754.738} C_VEL
LIN {X 0,Y 675.83,Z 820.614,A -85,B 0,C 180,E1 4757.722,E2 4757.722} C_VEL
LIN {X 0,Y 675.382,Z 838,A -85,B 0,C 180,E1 4760.961,E2 4760.961} C_VEL
LIN {X 0,Y 675.282,Z 849.595,A -85,B 0,C 180,E1 4764.201,E2 4764.201} C_VEL
LIN {X 0,Y 675.213,Z 855.945,A -85,B 0,C 180,E1 4767.424,E2 4767.424} C_VEL
LIN {X 0,Y 675.135,Z 857.433,A -85,B 0,C 180,E1 4769.996,E2 4769.996} C_VEL
LIN {X 0,Y 675.187,Z 855.836,A -85,B 0,C 180,E1 4772.569,E2 4772.569} C_VEL
LIN {X 0,Y 675.299,Z 849.361,A -85,B 0,C 180,E1 4775.791,E2 4775.791} C_VEL
LIN {X 0,Y 675.385,Z 837.644,A -85,B 0,C 180,E1 4779.032,E2 4779.032} C_VEL
LIN {X 0,Y 675.842,Z 819.975,A -85,B 0,C 180,E1 4782.284,E2 4782.284} C_VEL
LIN {X 0,Y 676.492,Z 797.636,A -85,B 0,C 180,E1 4785.255,E2 4785.255} C_VEL
LIN {X 0,Y 677.616,Z 769.747,A -85,B 0,C 180,E1 4788.057,E2 4788.057} C_VEL
LIN {X 0,Y 678.958,Z 738.323,A -85,B 0,C 180,E1 4790.435,E2 4790.435} C_VEL
LIN {X 0,Y 680.456,Z 702.525,A -85,B 0,C 180,E1 4792.459,E2 4792.459} C_VEL
LIN {X 0,Y 681.838,Z 665.638,A -85,B 0,C 180,E1 4793.963,E2 4793.963} C_VEL
LIN {X 0,Y 682.768,Z 628.011,A -85,B 0,C 180,E1 4794.974,E2 4794.974} C_VEL
LIN {X 0,Y 679.306,Z 615.168,A -85,B 0,C 180,E1 4795.367,E2 4795.367} C_VEL
LIN {X 0,Y 674.585,Z 601.31,A -85,B 0,C 180,E1 4795.784,E2 4795.784} C_VEL
LIN {X 0,Y 674.584,Z 601.31,A -85,B 0,C 180,E1 4801.425,E2 4801.425} C_VEL
LIN {X 0,Y 674.513,Z 601.31,A -85,B 0,C 180,E1 4806.051,E2 4806.051} C_VEL
LIN {X 0,Y 674.494,Z 601.31,A -85,B 0,C 180,E1 4810.647,E2 4810.647} C_VEL
LIN {X 0,Y 674.569,Z 601.31,A -85,B 0,C 180,E1 4815.882,E2 4815.882} C_VEL
LIN {X 0,Y 674.496,Z 601.31,A -85,B 0,C 180,E1 4821.036,E2 4821.036} C_VEL
LIN {X 0,Y 674.532,Z 601.31,A -85,B 0,C 180,E1 4826.209,E2 4826.209} C_VEL
LIN {X 0,Y 674.615,Z 601.31,A -85,B 0,C 180,E1 4831.866,E2 4831.866} C_VEL
LIN {X 0,Y 674.697,Z 601.31,A -85,B 0,C 180,E1 4837.028,E2 4837.028} C_VEL
LIN {X 0,Y 674.569,Z 601.31,A -85,B 0,C 180,E1 4840.846,E2 4840.846} C_VEL
LIN {X 0,Y 679.77,Z 620.607,A -85,B 0,C 180,E1 4841.232,E2 4841.232} C_VEL
LIN {X 0,Y 679.327,Z 690.727,A -85,B 0,C 180,E1 4842.104,E2 4842.104} C_VEL
LIN {X 0,Y 678.766,Z 724.384,A -85,B 0,C 180,E1 4843.01,E2 4843.01} C_VEL
LIN {X 0,Y 677.856,Z 755.644,A -85,B 0,C 180,E1 4844.353,E2 4844.353} C_VEL
LIN {X 0,Y 677.076,Z 784.015,A -85,B 0,C 180,E1 4846.121,E2 4846.121} C_VEL
LIN {X 0,Y 676.325,Z 808.044,A -85,B 0,C 180,E1 4848.208,E2 4848.208} C_VEL
LIN {X 0,Y 675.789,Z 828.883,A -85,B 0,C 180,E1 4850.748,E2 4850.748} C_VEL
LIN {X 0,Y 675.49,Z 844.411,A -85,B 0,C 180,E1 4853.563,E2 4853.563} C_VEL
LIN {X 0,Y 675.342,Z 853.111,A -85,B 0,C 180,E1 4856.143,E2 4856.143} C_VEL
LIN {X 0,Y 675.253,Z 857.279,A -85,B 0,C 180,E1 4858.716,E2 4858.716} C_VEL
LIN {X 0,Y 675.269,Z 857.229,A -85,B 0,C 180,E1 4861.287,E2 4861.287} C_VEL
LIN {X 0,Y 675.356,Z 852.976,A -85,B 0,C 180,E1 4863.86,E2 4863.86} C_VEL
LIN {X 0,Y 675.532,Z 842.704,A -85,B 0,C 180,E1 4866.763,E2 4866.763} C_VEL
LIN {X 0,Y 675.881,Z 827.014,A -85,B 0,C 180,E1 4869.482,E2 4869.482} C_VEL
LIN {X 0,Y 676.475,Z 806.063,A -85,B 0,C 180,E1 4871.957,E2 4871.957} C_VEL
LIN {X 0,Y 677.259,Z 781.548,A -85,B 0,C 180,E1 4874.006,E2 4874.006} C_VEL
LIN {X 0,Y 678.02,Z 752.054,A -85,B 0,C 180,E1 4875.77,E2 4875.77} C_VEL
LIN {X 0,Y 678.83,Z 719.759,A -85,B 0,C 180,E1 4877.075,E2 4877.075} C_VEL
LIN {X 0,Y 679.322,Z 688.373,A -85,B 0,C 180,E1 4877.862,E2 4877.862} C_VEL
LIN {X 0,Y 677.292,Z 675.775,A -85,B 0,C 180,E1 4878.126,E2 4878.126} C_VEL
LIN {X 0,Y 672.3,Z 657.131,A -85,B 0,C 180,E1 4878.515,E2 4878.515} C_VEL
LIN {X 0,Y 672.225,Z 654.964,A -85,B 0,C 180,E1 4878.544,E2 4878.544} C_VEL
LIN {X 0,Y 671.7,Z 616.92,A -85,B 0,C 180,E1 4879.042,E2 4879.042} C_VEL
LIN {X 0,Y 666.947,Z 601.31,A -85,B 0,C 180,E1 4879.455,E2 4879.455} C_VEL
LIN {X 0,Y 666.681,Z 601.31,A -85,B 0,C 180,E1 4884.627,E2 4884.627} C_VEL
LIN {X 0,Y 666.639,Z 601.31,A -85,B 0,C 180,E1 4889.997,E2 4889.997} C_VEL
LIN {X 0,Y 666.629,Z 601.31,A -85,B 0,C 180,E1 4895.096,E2 4895.096} C_VEL
LIN {X 0,Y 666.606,Z 601.31,A -85,B 0,C 180,E1 4899.519,E2 4899.519} C_VEL
LIN {X 0,Y 666.649,Z 601.31,A -85,B 0,C 180,E1 4904.786,E2 4904.786} C_VEL
LIN {X 0,Y 666.569,Z 601.31,A -85,B 0,C 180,E1 4910.6,E2 4910.6} C_VEL
LIN {X 0,Y 666.585,Z 601.444,A -85,B 0,C 180,E1 4915.465,E2 4915.465} C_VEL
LIN {X 0,Y 672.167,Z 614.816,A -85,B 0,C 180,E1 4915.82,E2 4915.82} C_VEL
LIN {X 0,Y 681.756,Z 634.986,A -85,B 0,C 180,E1 4916.555,E2 4916.555} C_VEL
LIN {X 0,Y 680.889,Z 708.393,A -85,B 0,C 180,E1 4917.531,E2 4917.531} C_VEL
LIN {X 0,Y 679.467,Z 748.659,A -85,B 0,C 180,E1 4918.497,E2 4918.497} C_VEL
LIN {X 0,Y 677.603,Z 791.115,A -85,B 0,C 180,E1 4920.03,E2 4920.03} C_VEL
LIN {X 0,Y 675.437,Z 830.897,A -85,B 0,C 180,E1 4922.008,E2 4922.008} C_VEL
LIN {X 0,Y 673.243,Z 867.765,A -85,B 0,C 180,E1 4924.391,E2 4924.391} C_VEL
LIN {X 0,Y 671.167,Z 902.493,A -85,B 0,C 180,E1 4927.26,E2 4927.26} C_VEL
LIN {X 0,Y 669.468,Z 934.567,A -85,B 0,C 180,E1 4930.674,E2 4930.674} C_VEL
LIN {X 0,Y 668.325,Z 961.208,A -85,B 0,C 180,E1 4934.381,E2 4934.381} C_VEL
LIN {X 0,Y 667.674,Z 981.63,A -85,B 0,C 180,E1 4938.218,E2 4938.218} C_VEL
LIN {X 0,Y 667.459,Z 994.244,A -85,B 0,C 180,E1 4941.518,E2 4941.518} C_VEL
LIN {X 0,Y 667.283,Z 1003.671,A -85,B 0,C 180,E1 4945.445,E2 4945.445} C_VEL
LIN {X 0,Y 667.328,Z 1007.169,A -85,B 0,C 180,E1 4948.703,E2 4948.703} C_VEL
LIN {X 0,Y 667.309,Z 1006.139,A -85,B 0,C 180,E1 4952.702,E2 4952.702} C_VEL
LIN {X 0,Y 667.272,Z 999.628,A -85,B 0,C 180,E1 4956.523,E2 4956.523} C_VEL
LIN {X 0,Y 667.468,Z 988.504,A -85,B 0,C 180,E1 4960.136,E2 4960.136} C_VEL
LIN {X 0,Y 667.854,Z 971.773,A -85,B 0,C 180,E1 4963.785,E2 4963.785} C_VEL
LIN {X 0,Y 668.58,Z 951.152,A -85,B 0,C 180,E1 4967.138,E2 4967.138} C_VEL
LIN {X 0,Y 669.97,Z 924.121,A -85,B 0,C 180,E1 4970.538,E2 4970.538} C_VEL
LIN {X 0,Y 671.911,Z 889.901,A -85,B 0,C 180,E1 4973.864,E2 4973.864} C_VEL
LIN {X 0,Y 674.227,Z 851.912,A -85,B 0,C 180,E1 4976.713,E2 4976.713} C_VEL
LIN {X 0,Y 676.502,Z 811.113,A -85,B 0,C 180,E1 4979.049,E2 4979.049} C_VEL
LIN {X 0,Y 678.577,Z 770.536,A -85,B 0,C 180,E1 4980.776,E2 4980.776} C_VEL
LIN {X 0,Y 680.337,Z 728.488,A -85,B 0,C 180,E1 4982.042,E2 4982.042} C_VEL
LIN {X 0,Y 681.292,Z 685.197,A -85,B 0,C 180,E1 4982.84,E2 4982.84} C_VEL
LIN {X 0,Y 681.148,Z 632.253,A -85,B 0,C 180,E1 4983.513,E2 4983.513} C_VEL
LIN {X 0,Y 666.89,Z 602.943,A -85,B 0,C 180,E1 4984.59,E2 4984.59} C_VEL
LIN {X 0,Y 666.75,Z 601.31,A -85,B 0,C 180,E1 4984.624,E2 4984.624} C_VEL
LIN {X 0,Y 666.565,Z 601.31,A -85,B 0,C 180,E1 4989.535,E2 4989.535} C_VEL
LIN {X 0,Y 666.622,Z 601.31,A -85,B 0,C 180,E1 4994.804,E2 4994.804} C_VEL
LIN {X 0,Y 666.581,Z 601.31,A -85,B 0,C 180,E1 5000.616,E2 5000.616} C_VEL
LIN {X 0,Y 666.533,Z 601.31,A -85,B 0,C 180,E1 5005.374,E2 5005.374} C_VEL
LIN {X 0,Y 666.619,Z 601.31,A -85,B 0,C 180,E1 5010.002,E2 5010.002} C_VEL
LIN {X 0,Y 666.755,Z 601.31,A -85,B 0,C 180,E1 5015.376,E2 5015.376} C_VEL
LIN {X 0,Y 666.801,Z 601.31,A -85,B 0,C 180,E1 5020.074,E2 5020.074} C_VEL
LIN {X 0,Y 666.861,Z 601.31,A -85,B 0,C 180,E1 5024.179,E2 5024.179} C_VEL
LIN {X 0,Y 666.942,Z 601.31,A -85,B 0,C 180,E1 5029.529,E2 5029.529} C_VEL
LIN {X 0,Y 667.013,Z 601.31,A -85,B 0,C 180,E1 5034.786,E2 5034.786} C_VEL
LIN {X 0,Y 667.108,Z 601.31,A -85,B 0,C 180,E1 5039.998,E2 5039.998} C_VEL
LIN {X 0,Y 667.215,Z 601.31,A -85,B 0,C 180,E1 5045.209,E2 5045.209} C_VEL
LIN {X 0,Y 666.914,Z 601.31,A -85,B 0,C 180,E1 5050.468,E2 5050.468} C_VEL
LIN {X 0,Y 666.888,Z 601.31,A -85,B 0,C 180,E1 5055.817,E2 5055.817} C_VEL
LIN {X 0,Y 666.837,Z 601.31,A -85,B 0,C 180,E1 5061.312,E2 5061.312} C_VEL
LIN {X 0,Y 666.748,Z 601.31,A -85,B 0,C 180,E1 5065.573,E2 5065.573} C_VEL
LIN {X 0,Y 666.629,Z 601.31,A -85,B 0,C 180,E1 5070.257,E2 5070.257} C_VEL
LIN {X 0,Y 666.583,Z 601.31,A -85,B 0,C 180,E1 5075.077,E2 5075.077} C_VEL
LIN {X 0,Y 666.587,Z 601.31,A -85,B 0,C 180,E1 5079.516,E2 5079.516} C_VEL
LIN {X 0,Y 666.656,Z 601.31,A -85,B 0,C 180,E1 5084.781,E2 5084.781} C_VEL
LIN {X 0,Y 666.575,Z 601.31,A -85,B 0,C 180,E1 5090.594,E2 5090.594} C_VEL
LIN {X 0,Y 666.566,Z 601.31,A -85,B 0,C 180,E1 5095.365,E2 5095.365} C_VEL
LIN {X 0,Y 666.644,Z 601.31,A -85,B 0,C 180,E1 5099.994,E2 5099.994} C_VEL
LIN {X 0,Y 666.922,Z 601.31,A -85,B 0,C 180,E1 5103.905,E2 5103.905} C_VEL
LIN {X 0,Y 675.543,Z 629.327,A -85,B 0,C 180,E1 5104.679,E2 5104.679} C_VEL
LIN {X 0,Y 674.421,Z 668.352,A -85,B 0,C 180,E1 5105.768,E2 5105.768} C_VEL
LIN {X 0,Y 672.92,Z 705.986,A -85,B 0,C 180,E1 5107.364,E2 5107.364} C_VEL
LIN {X 0,Y 671.332,Z 741.053,A -85,B 0,C 180,E1 5109.414,E2 5109.414} C_VEL
LIN {X 0,Y 669.793,Z 772.532,A -85,B 0,C 180,E1 5111.895,E2 5111.895} C_VEL
LIN {X 0,Y 668.689,Z 799.803,A -85,B 0,C 180,E1 5114.727,E2 5114.727} C_VEL
LIN {X 0,Y 667.972,Z 821.348,A -85,B 0,C 180,E1 5117.693,E2 5117.693} C_VEL
LIN {X 0,Y 667.513,Z 837.992,A -85,B 0,C 180,E1 5120.854,E2 5120.854} C_VEL
LIN {X 0,Y 667.382,Z 849.588,A -85,B 0,C 180,E1 5124.132,E2 5124.132} C_VEL
LIN {X 0,Y 667.32,Z 855.944,A -85,B 0,C 180,E1 5127.394,E2 5127.394} C_VEL
LIN {X 0,Y 667.235,Z 857.427,A -85,B 0,C 180,E1 5129.996,E2 5129.996} C_VEL
LIN {X 0,Y 667.286,Z 855.659,A -85,B 0,C 180,E1 5132.731,E2 5132.731} C_VEL
LIN {X 0,Y 667.4,Z 849.357,A -85,B 0,C 180,E1 5135.86,E2 5135.86} C_VEL
LIN {X 0,Y 667.518,Z 837.64,A -85,B 0,C 180,E1 5139.139,E2 5139.139} C_VEL
LIN {X 0,Y 667.988,Z 820.789,A -85,B 0,C 180,E1 5142.307,E2 5142.307} C_VEL
LIN {X 0,Y 668.754,Z 797.634,A -85,B 0,C 180,E1 5145.436,E2 5145.436} C_VEL
LIN {X 0,Y 669.972,Z 769.847,A -85,B 0,C 180,E1 5148.261,E2 5148.261} C_VEL
LIN {X 0,Y 671.454,Z 738.318,A -85,B 0,C 180,E1 5150.674,E2 5150.674} C_VEL
LIN {X 0,Y 673.114,Z 701.921,A -85,B 0,C 180,E1 5152.748,E2 5152.748} C_VEL
LIN {X 0,Y 674.61,Z 664.338,A -85,B 0,C 180,E1 5154.281,E2 5154.281} C_VEL
LIN {X 0,Y 674.865,Z 625.19,A -85,B 0,C 180,E1 5155.336,E2 5155.336} C_VEL
LIN {X 0,Y 666.658,Z 601.31,A -85,B 0,C 180,E1 5156.087,E2 5156.087} C_VEL
LIN {X 0,Y 666.687,Z 601.31,A -85,B 0,C 180,E1 5161.511,E2 5161.511} C_VEL
LIN {X 0,Y 666.599,Z 601.31,A -85,B 0,C 180,E1 5166.223,E2 5166.223} C_VEL
LIN {X 0,Y 666.605,Z 601.31,A -85,B 0,C 180,E1 5171.418,E2 5171.418} C_VEL
LIN {X 0,Y 666.552,Z 601.31,A -85,B 0,C 180,E1 5176.666,E2 5176.666} C_VEL
LIN {X 0,Y 666.569,Z 601.31,A -85,B 0,C 180,E1 5182.151,E2 5182.151} C_VEL
LIN {X 0,Y 666.655,Z 601.31,A -85,B 0,C 180,E1 5187.234,E2 5187.234} C_VEL
LIN {X 0,Y 666.739,Z 601.31,A -85,B 0,C 180,E1 5192.975,E2 5192.975} C_VEL
LIN {X 0,Y 666.782,Z 601.31,A -85,B 0,C 180,E1 5197.282,E2 5197.282} C_VEL
LIN {X 0,Y 666.703,Z 601.31,A -85,B 0,C 180,E1 5200.58,E2 5200.58} C_VEL
LIN {X 0,Y 672.364,Z 622.331,A -85,B 0,C 180,E1 5201.023,E2 5201.023} C_VEL
LIN {X 0,Y 671.763,Z 693.025,A -85,B 0,C 180,E1 5201.938,E2 5201.938} C_VEL
LIN {X 0,Y 671.177,Z 727.097,A -85,B 0,C 180,E1 5202.897,E2 5202.897} C_VEL
LIN {X 0,Y 670.198,Z 759.273,A -85,B 0,C 180,E1 5204.348,E2 5204.348} C_VEL
LIN {X 0,Y 669.283,Z 787.982,A -85,B 0,C 180,E1 5206.228,E2 5206.228} C_VEL
LIN {X 0,Y 668.494,Z 811.788,A -85,B 0,C 180,E1 5208.399,E2 5208.399} C_VEL
LIN {X 0,Y 667.95,Z 831.1,A -85,B 0,C 180,E1 5210.867,E2 5210.867} C_VEL
LIN {X 0,Y 667.682,Z 845.243,A -85,B 0,C 180,E1 5213.488,E2 5213.488} C_VEL
LIN {X 0,Y 667.51,Z 854.046,A -85,B 0,C 180,E1 5216.098,E2 5216.098} C_VEL
LIN {X 0,Y 667.432,Z 858.288,A -85,B 0,C 180,E1 5218.701,E2 5218.701} C_VEL
LIN {X 0,Y 667.447,Z 858.28,A -85,B 0,C 180,E1 5221.302,E2 5221.302} C_VEL
LIN {X 0,Y 667.548,Z 854.037,A -85,B 0,C 180,E1 5223.905,E2 5223.905} C_VEL
LIN {X 0,Y 667.749,Z 843.731,A -85,B 0,C 180,E1 5226.842,E2 5226.842} C_VEL
LIN {X 0,Y 668.128,Z 827.973,A -85,B 0,C 180,E1 5229.593,E2 5229.593} C_VEL
LIN {X 0,Y 668.773,Z 806.907,A -85,B 0,C 180,E1 5232.096,E2 5232.096} C_VEL
LIN {X 0,Y 669.612,Z 781.225,A -85,B 0,C 180,E1 5234.244,E2 5234.244} C_VEL
LIN {X 0,Y 670.485,Z 751.448,A -85,B 0,C 180,E1 5236.007,E2 5236.007} C_VEL
LIN {X 0,Y 671.355,Z 718.912,A -85,B 0,C 180,E1 5237.313,E2 5237.313} C_VEL
LIN {X 0,Y 671.964,Z 684.549,A -85,B 0,C 180,E1 5238.145,E2 5238.145} C_VEL
LIN {X 0,Y 672.225,Z 654.964,A -85,B 0,C 180,E1 5238.544,E2 5238.544} C_VEL
LIN {X 0,Y 669.125,Z 638.153,A -85,B 0,C 180,E1 5238.857,E2 5238.857} C_VEL
LIN {X 0,Y 665.07,Z 621.465,A -85,B 0,C 180,E1 5239.21,E2 5239.21} C_VEL
LIN {X 0,Y 659.014,Z 601.31,A -85,B 0,C 180,E1 5239.739,E2 5239.739} C_VEL
LIN {X 0,Y 658.784,Z 601.31,A -85,B 0,C 180,E1 5244.453,E2 5244.453} C_VEL
LIN {X 0,Y 658.744,Z 601.31,A -85,B 0,C 180,E1 5249.074,E2 5249.074} C_VEL
LIN {X 0,Y 658.727,Z 601.31,A -85,B 0,C 180,E1 5254.105,E2 5254.105} C_VEL
LIN {X 0,Y 658.673,Z 601.31,A -85,B 0,C 180,E1 5258.55,E2 5258.55} C_VEL
LIN {X 0,Y 658.741,Z 601.31,A -85,B 0,C 180,E1 5263.624,E2 5263.624} C_VEL
LIN {X 0,Y 658.583,Z 601.31,A -85,B 0,C 180,E1 5269.385,E2 5269.385} C_VEL
LIN {X 0,Y 658.672,Z 601.31,A -85,B 0,C 180,E1 5275.172,E2 5275.172} C_VEL
LIN {X 0,Y 665.146,Z 617.88,A -85,B 0,C 180,E1 5275.597,E2 5275.597} C_VEL
LIN {X 0,Y 675.125,Z 638.669,A -85,B 0,C 180,E1 5276.23,E2 5276.23} C_VEL
LIN {X 0,Y 674.216,Z 708.793,A -85,B 0,C 180,E1 5277.177,E2 5277.177} C_VEL
LIN {X 0,Y 672.655,Z 749.376,A -85,B 0,C 180,E1 5278.165,E2 5278.165} C_VEL
LIN {X 0,Y 670.59,Z 792.432,A -85,B 0,C 180,E1 5279.742,E2 5279.742} C_VEL
LIN {X 0,Y 668.222,Z 832.627,A -85,B 0,C 180,E1 5281.783,E2 5281.783} C_VEL
LIN {X 0,Y 665.831,Z 869.039,A -85,B 0,C 180,E1 5284.185,E2 5284.185} C_VEL
LIN {X 0,Y 663.537,Z 904.257,A -85,B 0,C 180,E1 5287.161,E2 5287.161} C_VEL
LIN {X 0,Y 661.762,Z 934.567,A -85,B 0,C 180,E1 5290.44,E2 5290.44} C_VEL
LIN {X 0,Y 660.518,Z 961.807,A -85,B 0,C 180,E1 5294.287,E2 5294.287} C_VEL
LIN {X 0,Y 659.828,Z 981.629,A -85,B 0,C 180,E1 5298.076,E2 5298.076} C_VEL
LIN {X 0,Y 659.573,Z 994.571,A -85,B 0,C 180,E1 5301.529,E2 5301.529} C_VEL
LIN {X 0,Y 659.403,Z 1003.671,A -85,B 0,C 180,E1 5305.391,E2 5305.391} C_VEL
LIN {X 0,Y 659.433,Z 1007.168,A -85,B 0,C 180,E1 5308.687,E2 5308.687} C_VEL
LIN {X 0,Y 659.449,Z 1006.214,A -85,B 0,C 180,E1 5312.638,E2 5312.638} C_VEL
LIN {X 0,Y 659.477,Z 1001.189,A -85,B 0,C 180,E1 5315.938,E2 5315.938} C_VEL
LIN {X 0,Y 659.579,Z 989.706,A -85,B 0,C 180,E1 5319.925,E2 5319.925} C_VEL
LIN {X 0,Y 659.972,Z 973.52,A -85,B 0,C 180,E1 5323.615,E2 5323.615} C_VEL
LIN {X 0,Y 660.793,Z 952.352,A -85,B 0,C 180,E1 5327.175,E2 5327.175} C_VEL
LIN {X 0,Y 662.379,Z 924.071,A -85,B 0,C 180,E1 5330.789,E2 5330.789} C_VEL
LIN {X 0,Y 664.4,Z 890.604,A -85,B 0,C 180,E1 5334.089,E2 5334.089} C_VEL
LIN {X 0,Y 666.948,Z 851.91,A -85,B 0,C 180,E1 5337.028,E2 5337.028} C_VEL
LIN {X 0,Y 669.504,Z 810.546,A -85,B 0,C 180,E1 5339.413,E2 5339.413} C_VEL
LIN {X 0,Y 671.825,Z 768.706,A -85,B 0,C 180,E1 5341.191,E2 5341.191} C_VEL
LIN {X 0,Y 673.621,Z 728.491,A -85,B 0,C 180,E1 5342.4,E2 5342.4} C_VEL
LIN {X 0,Y 674.685,Z 684.34,A -85,B 0,C 180,E1 5343.216,E2 5343.216} C_VEL
LIN {X 0,Y 674.761,Z 635.427,A -85,B 0,C 180,E1 5343.829,E2 5343.829} C_VEL
LIN {X 0,Y 658.928,Z 602.71,A -85,B 0,C 180,E1 5344.982,E2 5344.982} C_VEL
LIN {X 0,Y 658.782,Z 601.31,A -85,B 0,C 180,E1 5345.104,E2 5345.104} C_VEL
LIN {X 0,Y 658.623,Z 601.31,A -85,B 0,C 180,E1 5350.619,E2 5350.619} C_VEL
LIN {X 0,Y 658.662,Z 601.31,A -85,B 0,C 180,E1 5355.496,E2 5355.496} C_VEL
LIN {X 0,Y 658.597,Z 601.31,A -85,B 0,C 180,E1 5359.904,E2 5359.904} C_VEL
LIN {X 0,Y 658.635,Z 601.31,A -85,B 0,C 180,E1 5364.898,E2 5364.898} C_VEL
LIN {X 0,Y 658.734,Z 601.31,A -85,B 0,C 180,E1 5369.605,E2 5369.605} C_VEL
LIN {X 0,Y 658.827,Z 601.31,A -85,B 0,C 180,E1 5374.093,E2 5374.093} C_VEL
LIN {X 0,Y 658.876,Z 601.31,A -85,B 0,C 180,E1 5378.414,E2 5378.414} C_VEL
LIN {X 0,Y 658.946,Z 601.31,A -85,B 0,C 180,E1 5383.984,E2 5383.984} C_VEL
LIN {X 0,Y 659.018,Z 601.31,A -85,B 0,C 180,E1 5389.402,E2 5389.402} C_VEL
LIN {X 0,Y 659.109,Z 601.31,A -85,B 0,C 180,E1 5394.723,E2 5394.723} C_VEL
LIN {X 0,Y 659.225,Z 601.31,A -85,B 0,C 180,E1 5399.998,E2 5399.998} C_VEL
LIN {X 0,Y 659.293,Z 601.31,A -85,B 0,C 180,E1 5405.272,E2 5405.272} C_VEL
LIN {X 0,Y 658.999,Z 601.31,A -85,B 0,C 180,E1 5410.595,E2 5410.595} C_VEL
LIN {X 0,Y 658.972,Z 601.31,A -85,B 0,C 180,E1 5416.012,E2 5416.012} C_VEL
LIN {X 0,Y 658.897,Z 601.31,A -85,B 0,C 180,E1 5421.582,E2 5421.582} C_VEL
LIN {X 0,Y 658.803,Z 601.31,A -85,B 0,C 180,E1 5426.229,E2 5426.229} C_VEL
LIN {X 0,Y 658.738,Z 601.31,A -85,B 0,C 180,E1 5431.931,E2 5431.931} C_VEL
LIN {X 0,Y 658.718,Z 601.31,A -85,B 0,C 180,E1 5436.72,E2 5436.72} C_VEL
LIN {X 0,Y 658.711,Z 601.31,A -85,B 0,C 180,E1 5442.596,E2 5442.596} C_VEL
LIN {X 0,Y 658.604,Z 601.31,A -85,B 0,C 180,E1 5447.393,E2 5447.393} C_VEL
LIN {X 0,Y 658.625,Z 601.31,A -85,B 0,C 180,E1 5451.595,E2 5451.595} C_VEL
LIN {X 0,Y 658.667,Z 601.31,A -85,B 0,C 180,E1 5456.485,E2 5456.485} C_VEL
LIN {X 0,Y 658.747,Z 601.31,A -85,B 0,C 180,E1 5461.113,E2 5461.113} C_VEL
LIN {X 0,Y 658.966,Z 601.31,A -85,B 0,C 180,E1 5463.613,E2 5463.613} C_VEL
LIN {X 0,Y 668.203,Z 629.549,A -85,B 0,C 180,E1 5464.431,E2 5464.431} C_VEL
LIN {X 0,Y 667.126,Z 668.327,A -85,B 0,C 180,E1 5465.502,E2 5465.502} C_VEL
LIN {X 0,Y 665.595,Z 704.879,A -85,B 0,C 180,E1 5467.044,E2 5467.044} C_VEL
LIN {X 0,Y 663.884,Z 739.783,A -85,B 0,C 180,E1 5469.088,E2 5469.088} C_VEL
LIN {X 0,Y 662.277,Z 771.017,A -85,B 0,C 180,E1 5471.54,E2 5471.54} C_VEL
LIN {X 0,Y 660.954,Z 799.647,A -85,B 0,C 180,E1 5474.527,E2 5474.527} C_VEL
LIN {X 0,Y 660.136,Z 821.744,A -85,B 0,C 180,E1 5477.613,E2 5477.613} C_VEL
LIN {X 0,Y 659.624,Z 838.776,A -85,B 0,C 180,E1 5480.932,E2 5480.932} C_VEL
LIN {X 0,Y 659.489,Z 849.581,A -85,B 0,C 180,E1 5484.062,E2 5484.062} C_VEL
LIN {X 0,Y 659.439,Z 855.943,A -85,B 0,C 180,E1 5487.362,E2 5487.362} C_VEL
LIN {X 0,Y 659.341,Z 857.421,A -85,B 0,C 180,E1 5489.996,E2 5489.996} C_VEL
LIN {X 0,Y 659.434,Z 855.837,A -85,B 0,C 180,E1 5492.63,E2 5492.63} C_VEL
LIN {X 0,Y 659.514,Z 849.353,A -85,B 0,C 180,E1 5495.931,E2 5495.931} C_VEL
LIN {X 0,Y 659.669,Z 837.636,A -85,B 0,C 180,E1 5499.249,E2 5499.249} C_VEL
LIN {X 0,Y 660.153,Z 821.195,A -85,B 0,C 180,E1 5502.391,E2 5502.391} C_VEL
LIN {X 0,Y 660.97,Z 798.911,A -85,B 0,C 180,E1 5505.47,E2 5505.47} C_VEL
LIN {X 0,Y 662.274,Z 771.299,A -85,B 0,C 180,E1 5508.343,E2 5508.343} C_VEL
LIN {X 0,Y 663.819,Z 741.19,A -85,B 0,C 180,E1 5510.73,E2 5510.73} C_VEL
LIN {X 0,Y 665.498,Z 706.841,A -85,B 0,C 180,E1 5512.768,E2 5512.768} C_VEL
LIN {X 0,Y 667.083,Z 670.023,A -85,B 0,C 180,E1 5514.345,E2 5514.345} C_VEL
LIN {X 0,Y 668.182,Z 631.089,A -85,B 0,C 180,E1 5515.445,E2 5515.445} C_VEL
LIN {X 0,Y 658.742,Z 601.31,A -85,B 0,C 180,E1 5516.351,E2 5516.351} C_VEL
LIN {X 0,Y 658.769,Z 601.31,A -85,B 0,C 180,E1 5521.934,E2 5521.934} C_VEL
LIN {X 0,Y 658.685,Z 601.31,A -85,B 0,C 180,E1 5526.729,E2 5526.729} C_VEL
LIN {X 0,Y 658.726,Z 601.31,A -85,B 0,C 180,E1 5532.618,E2 5532.618} C_VEL
LIN {X 0,Y 658.59,Z 601.31,A -85,B 0,C 180,E1 5537.405,E2 5537.405} C_VEL
LIN {X 0,Y 658.612,Z 601.31,A -85,B 0,C 180,E1 5541.611,E2 5541.611} C_VEL
LIN {X 0,Y 658.667,Z 601.31,A -85,B 0,C 180,E1 5546.499,E2 5546.499} C_VEL
LIN {X 0,Y 658.726,Z 601.31,A -85,B 0,C 180,E1 5551.124,E2 5551.124} C_VEL
LIN {X 0,Y 658.886,Z 601.31,A -85,B 0,C 180,E1 5555.555,E2 5555.555} C_VEL
LIN {X 0,Y 658.749,Z 601.31,A -85,B 0,C 180,E1 5560.326,E2 5560.326} C_VEL
LIN {X 0,Y 664.911,Z 623.511,A -85,B 0,C 180,E1 5560.806,E2 5560.806} C_VEL
LIN {X 0,Y 664.344,Z 691.423,A -85,B 0,C 180,E1 5561.686,E2 5561.686} C_VEL
LIN {X 0,Y 663.639,Z 726.176,A -85,B 0,C 180,E1 5562.654,E2 5562.654} C_VEL
LIN {X 0,Y 662.618,Z 758.071,A -85,B 0,C 180,E1 5564.079,E2 5564.079} C_VEL
LIN {X 0,Y 661.657,Z 786.642,A -85,B 0,C 180,E1 5565.923,E2 5565.923} C_VEL
LIN {X 0,Y 660.816,Z 810.802,A -85,B 0,C 180,E1 5568.095,E2 5568.095} C_VEL
LIN {X 0,Y 660.203,Z 831.317,A -85,B 0,C 180,E1 5570.684,E2 5570.684} C_VEL
LIN {X 0,Y 659.857,Z 846.077,A -85,B 0,C 180,E1 5573.41,E2 5573.41} C_VEL
LIN {X 0,Y 659.689,Z 854.965,A -85,B 0,C 180,E1 5576.051,E2 5576.051} C_VEL
LIN {X 0,Y 659.597,Z 859.29,A -85,B 0,C 180,E1 5578.686,E2 5578.686} C_VEL
LIN {X 0,Y 659.619,Z 859.331,A -85,B 0,C 180,E1 5581.318,E2 5581.318} C_VEL
LIN {X 0,Y 659.734,Z 855.098,A -85,B 0,C 180,E1 5583.952,E2 5583.952} C_VEL
LIN {X 0,Y 659.961,Z 844.766,A -85,B 0,C 180,E1 5586.923,E2 5586.923} C_VEL
LIN {X 0,Y 660.395,Z 829.034,A -85,B 0,C 180,E1 5589.691,E2 5589.691} C_VEL
LIN {X 0,Y 661.086,Z 807.943,A -85,B 0,C 180,E1 5592.218,E2 5592.218} C_VEL
LIN {X 0,Y 661.981,Z 781.894,A -85,B 0,C 180,E1 5594.412,E2 5594.412} C_VEL
LIN {X 0,Y 662.928,Z 751.843,A -85,B 0,C 180,E1 5596.201,E2 5596.201} C_VEL
LIN {X 0,Y 663.859,Z 719.386,A -85,B 0,C 180,E1 5597.515,E2 5597.515} C_VEL
LIN {X 0,Y 664.544,Z 682.95,A -85,B 0,C 180,E1 5598.398,E2 5598.398} C_VEL
LIN {X 0,Y 665.07,Z 621.465,A -85,B 0,C 180,E1 5599.21,E2 5599.21} C_VEL
LIN {X 0,Y 660.942,Z 614.382,A -85,B 0,C 180,E1 5599.455,E2 5599.455} C_VEL
LIN {X 0,Y 652.089,Z 605.298,A -85,B 0,C 180,E1 5599.911,E2 5599.911} C_VEL
LIN {X 0,Y 651.553,Z 603.959,A -85,B 0,C 180,E1 5599.952,E2 5599.952} C_VEL
LIN {X 0,Y 651.065,Z 601.31,A -85,B 0,C 180,E1 5600.014,E2 5600.014} C_VEL
LIN {X 0,Y 650.858,Z 601.31,A -85,B 0,C 180,E1 5604.789,E2 5604.789} C_VEL
LIN {X 0,Y 650.841,Z 601.31,A -85,B 0,C 180,E1 5609.263,E2 5609.263} C_VEL
LIN {X 0,Y 650.848,Z 601.31,A -85,B 0,C 180,E1 5613.962,E2 5613.962} C_VEL
LIN {X 0,Y 650.738,Z 601.31,A -85,B 0,C 180,E1 5618.945,E2 5618.945} C_VEL
LIN {X 0,Y 650.837,Z 601.31,A -85,B 0,C 180,E1 5624.291,E2 5624.291} C_VEL
LIN {X 0,Y 650.656,Z 601.31,A -85,B 0,C 180,E1 5630.206,E2 5630.206} C_VEL
LIN {X 0,Y 650.851,Z 602.031,A -85,B 0,C 180,E1 5634.885,E2 5634.885} C_VEL
LIN {X 0,Y 658.65,Z 621.696,A -85,B 0,C 180,E1 5635.397,E2 5635.397} C_VEL
LIN {X 0,Y 667.973,Z 639.309,A -85,B 0,C 180,E1 5635.942,E2 5635.942} C_VEL
LIN {X 0,Y 667.494,Z 708.5,A -85,B 0,C 180,E1 5636.818,E2 5636.818} C_VEL
LIN {X 0,Y 665.967,Z 748.208,A -85,B 0,C 180,E1 5637.767,E2 5637.767} C_VEL
LIN {X 0,Y 663.728,Z 791.45,A -85,B 0,C 180,E1 5639.352,E2 5639.352} C_VEL
LIN {X 0,Y 661.076,Z 831.931,A -85,B 0,C 180,E1 5641.408,E2 5641.408} C_VEL
LIN {X 0,Y 658.578,Z 867.809,A -85,B 0,C 180,E1 5643.782,E2 5643.782} C_VEL
LIN {X 0,Y 656.165,Z 902.679,A -85,B 0,C 180,E1 5646.729,E2 5646.729} C_VEL
LIN {X 0,Y 654.075,Z 934.566,A -85,B 0,C 180,E1 5650.2,E2 5650.2} C_VEL
LIN {X 0,Y 652.801,Z 960.145,A -85,B 0,C 180,E1 5653.831,E2 5653.831} C_VEL
LIN {X 0,Y 652.012,Z 979.162,A -85,B 0,C 180,E1 5657.384,E2 5657.384} C_VEL
LIN {X 0,Y 651.687,Z 993.355,A -85,B 0,C 180,E1 5661.026,E2 5661.026} C_VEL
LIN {X 0,Y 651.584,Z 1002.467,A -85,B 0,C 180,E1 5664.667,E2 5664.667} C_VEL
LIN {X 0,Y 651.554,Z 1007.168,A -85,B 0,C 180,E1 5668.671,E2 5668.671} C_VEL
LIN {X 0,Y 651.546,Z 1006.214,A -85,B 0,C 180,E1 5672.67,E2 5672.67} C_VEL
LIN {X 0,Y 651.59,Z 1001.189,A -85,B 0,C 180,E1 5676.01,E2 5676.01} C_VEL
LIN {X 0,Y 651.711,Z 989.706,A -85,B 0,C 180,E1 5680.046,E2 5680.046} C_VEL
LIN {X 0,Y 652.14,Z 973.519,A -85,B 0,C 180,E1 5683.781,E2 5683.781} C_VEL
LIN {X 0,Y 653.068,Z 952.351,A -85,B 0,C 180,E1 5687.384,E2 5687.384} C_VEL
LIN {X 0,Y 654.764,Z 924.24,A -85,B 0,C 180,E1 5691.024,E2 5691.024} C_VEL
LIN {X 0,Y 656.982,Z 890.604,A -85,B 0,C 180,E1 5694.379,E2 5694.379} C_VEL
LIN {X 0,Y 659.73,Z 851.908,A -85,B 0,C 180,E1 5697.349,E2 5697.349} C_VEL
LIN {X 0,Y 662.532,Z 809.909,A -85,B 0,C 180,E1 5699.789,E2 5699.789} C_VEL
LIN {X 0,Y 665.026,Z 767.136,A -85,B 0,C 180,E1 5701.607,E2 5701.607} C_VEL
LIN {X 0,Y 666.927,Z 726.466,A -85,B 0,C 180,E1 5702.811,E2 5702.811} C_VEL
LIN {X 0,Y 667.904,Z 681.454,A -85,B 0,C 180,E1 5703.598,E2 5703.598} C_VEL
LIN {X 0,Y 667.471,Z 637.122,A -85,B 0,C 180,E1 5704.152,E2 5704.152} C_VEL
LIN {X 0,Y 650.992,Z 602.721,A -85,B 0,C 180,E1 5705.38,E2 5705.38} C_VEL
LIN {X 0,Y 650.833,Z 601.31,A -85,B 0,C 180,E1 5705.443,E2 5705.443} C_VEL
LIN {X 0,Y 650.726,Z 601.31,A -85,B 0,C 180,E1 5710.695,E2 5710.695} C_VEL
LIN {X 0,Y 650.746,Z 601.31,A -85,B 0,C 180,E1 5715.701,E2 5715.701} C_VEL
LIN {X 0,Y 650.661,Z 601.31,A -85,B 0,C 180,E1 5721.05,E2 5721.05} C_VEL
LIN {X 0,Y 650.716,Z 601.31,A -85,B 0,C 180,E1 5726.03,E2 5726.03} C_VEL
LIN {X 0,Y 650.844,Z 601.31,A -85,B 0,C 180,E1 5730.737,E2 5730.737} C_VEL
LIN {X 0,Y 650.927,Z 601.31,A -85,B 0,C 180,E1 5735.232,E2 5735.232} C_VEL
LIN {X 0,Y 650.969,Z 601.31,A -85,B 0,C 180,E1 5739.568,E2 5739.568} C_VEL
LIN {X 0,Y 651.022,Z 601.31,A -85,B 0,C 180,E1 5743.784,E2 5743.784} C_VEL
LIN {X 0,Y 651.096,Z 601.31,A -85,B 0,C 180,E1 5749.271,E2 5749.271} C_VEL
LIN {X 0,Y 651.232,Z 601.31,A -85,B 0,C 180,E1 5754.659,E2 5754.659} C_VEL
LIN {X 0,Y 651.326,Z 601.31,A -85,B 0,C 180,E1 5759.998,E2 5759.998} C_VEL
LIN {X 0,Y 651.386,Z 601.31,A -85,B 0,C 180,E1 5765.336,E2 5765.336} C_VEL
LIN {X 0,Y 651.087,Z 601.31,A -85,B 0,C 180,E1 5770.726,E2 5770.726} C_VEL
LIN {X 0,Y 651.051,Z 601.31,A -85,B 0,C 180,E1 5776.212,E2 5776.212} C_VEL
LIN {X 0,Y 651.009,Z 601.31,A -85,B 0,C 180,E1 5781.4,E2 5781.4} C_VEL
LIN {X 0,Y 650.922,Z 601.31,A -85,B 0,C 180,E1 5786.241,E2 5786.241} C_VEL
LIN {X 0,Y 650.816,Z 601.31,A -85,B 0,C 180,E1 5790.801,E2 5790.801} C_VEL
LIN {X 0,Y 650.784,Z 601.31,A -85,B 0,C 180,E1 5795.585,E2 5795.585} C_VEL
LIN {X 0,Y 650.747,Z 601.31,A -85,B 0,C 180,E1 5800.676,E2 5800.676} C_VEL
LIN {X 0,Y 650.773,Z 601.31,A -85,B 0,C 180,E1 5805.689,E2 5805.689} C_VEL
LIN {X 0,Y 650.671,Z 601.31,A -85,B 0,C 180,E1 5811.038,E2 5811.038} C_VEL
LIN {X 0,Y 650.786,Z 601.31,A -85,B 0,C 180,E1 5816.024,E2 5816.024} C_VEL
LIN {X 0,Y 650.844,Z 601.31,A -85,B 0,C 180,E1 5820.728,E2 5820.728} C_VEL
LIN {X 0,Y 651.085,Z 602.047,A -85,B 0,C 180,E1 5823.374,E2 5823.374} C_VEL
LIN {X 0,Y 660.829,Z 631.304,A -85,B 0,C 180,E1 5824.217,E2 5824.217} C_VEL
LIN {X 0,Y 659.732,Z 668.942,A -85,B 0,C 180,E1 5825.27,E2 5825.27} C_VEL
LIN {X 0,Y 658.185,Z 704.678,A -85,B 0,C 180,E1 5826.778,E2 5826.778} C_VEL
LIN {X 0,Y 656.434,Z 739.447,A -85,B 0,C 180,E1 5828.818,E2 5828.818} C_VEL
LIN {X 0,Y 654.694,Z 770.409,A -85,B 0,C 180,E1 5831.262,E2 5831.262} C_VEL
LIN {X 0,Y 653.295,Z 798.313,A -85,B 0,C 180,E1 5834.182,E2 5834.182} C_VEL
LIN {X 0,Y 652.307,Z 821.25,A -85,B 0,C 180,E1 5837.377,E2 5837.377} C_VEL
LIN {X 0,Y 651.764,Z 837.975,A -85,B 0,C 180,E1 5840.631,E2 5840.631} C_VEL
LIN {X 0,Y 651.606,Z 849.574,A -85,B 0,C 180,E1 5843.99,E2 5843.99} C_VEL
LIN {X 0,Y 651.535,Z 855.942,A -85,B 0,C 180,E1 5847.33,E2 5847.33} C_VEL
LIN {X 0,Y 651.472,Z 857.247,A -85,B 0,C 180,E1 5850.963,E2 5850.963} C_VEL
LIN {X 0,Y 651.573,Z 853.896,A -85,B 0,C 180,E1 5853.997,E2 5853.997} C_VEL
LIN {X 0,Y 651.717,Z 845.313,A -85,B 0,C 180,E1 5857.343,E2 5857.343} C_VEL
LIN {X 0,Y 651.993,Z 831.297,A -85,B 0,C 180,E1 5860.711,E2 5860.711} C_VEL
LIN {X 0,Y 652.707,Z 812.1,A -85,B 0,C 180,E1 5863.933,E2 5863.933} C_VEL
LIN {X 0,Y 653.85,Z 787.017,A -85,B 0,C 180,E1 5867.008,E2 5867.008} C_VEL
LIN {X 0,Y 655.444,Z 757.421,A -85,B 0,C 180,E1 5869.757,E2 5869.757} C_VEL
LIN {X 0,Y 657.132,Z 725.758,A -85,B 0,C 180,E1 5871.978,E2 5871.978} C_VEL
LIN {X 0,Y 658.906,Z 688.046,A -85,B 0,C 180,E1 5873.906,E2 5873.906} C_VEL
LIN {X 0,Y 660.348,Z 649.829,A -85,B 0,C 180,E1 5875.238,E2 5875.238} C_VEL
LIN {X 0,Y 660.194,Z 629.226,A -85,B 0,C 180,E1 5875.763,E2 5875.763} C_VEL
LIN {X 0,Y 650.822,Z 601.31,A -85,B 0,C 180,E1 5876.623,E2 5876.623} C_VEL
LIN {X 0,Y 650.849,Z 601.31,A -85,B 0,C 180,E1 5880.804,E2 5880.804} C_VEL
LIN {X 0,Y 650.783,Z 601.31,A -85,B 0,C 180,E1 5885.592,E2 5885.592} C_VEL
LIN {X 0,Y 650.729,Z 601.31,A -85,B 0,C 180,E1 5890.686,E2 5890.686} C_VEL
LIN {X 0,Y 650.782,Z 601.31,A -85,B 0,C 180,E1 5895.709,E2 5895.709} C_VEL
LIN {X 0,Y 650.657,Z 601.31,A -85,B 0,C 180,E1 5901.054,E2 5901.054} C_VEL
LIN {X 0,Y 650.787,Z 601.31,A -85,B 0,C 180,E1 5906.039,E2 5906.039} C_VEL
LIN {X 0,Y 650.824,Z 601.31,A -85,B 0,C 180,E1 5910.74,E2 5910.74} C_VEL
LIN {X 0,Y 650.961,Z 601.31,A -85,B 0,C 180,E1 5915.238,E2 5915.238} C_VEL
LIN {X 0,Y 650.838,Z 601.31,A -85,B 0,C 180,E1 5920.039,E2 5920.039} C_VEL
LIN {X 0,Y 657.499,Z 624.752,A -85,B 0,C 180,E1 5920.582,E2 5920.582} C_VEL
LIN {X 0,Y 656.792,Z 693.66,A -85,B 0,C 180,E1 5921.512,E2 5921.512} C_VEL
LIN {X 0,Y 656.043,Z 728.77,A -85,B 0,C 180,E1 5922.533,E2 5922.533} C_VEL
LIN {X 0,Y 654.956,Z 759.964,A -85,B 0,C 180,E1 5923.974,E2 5923.974} C_VEL
LIN {X 0,Y 653.923,Z 789.231,A -85,B 0,C 180,E1 5925.924,E2 5925.924} C_VEL
LIN {X 0,Y 653.022,Z 812.979,A -85,B 0,C 180,E1 5928.121,E2 5928.121} C_VEL
LIN {X 0,Y 652.359,Z 833.509,A -85,B 0,C 180,E1 5930.799,E2 5930.799} C_VEL
LIN {X 0,Y 652.014,Z 848.267,A -85,B 0,C 180,E1 5933.666,E2 5933.666} C_VEL
LIN {X 0,Y 651.854,Z 857.418,A -85,B 0,C 180,E1 5936.671,E2 5936.671} C_VEL
LIN {X 0,Y 651.771,Z 860.28,A -85,B 0,C 180,E1 5938.67,E2 5938.67} C_VEL
LIN {X 0,Y 651.798,Z 860.028,A -85,B 0,C 180,E1 5941.744,E2 5941.744} C_VEL
LIN {X 0,Y 651.976,Z 854.373,A -85,B 0,C 180,E1 5944.666,E2 5944.666} C_VEL
LIN {X 0,Y 652.246,Z 842.607,A -85,B 0,C 180,E1 5947.676,E2 5947.676} C_VEL
LIN {X 0,Y 652.81,Z 826.029,A -85,B 0,C 180,E1 5950.362,E2 5950.362} C_VEL
LIN {X 0,Y 653.529,Z 803.829,A -85,B 0,C 180,E1 5952.842,E2 5952.842} C_VEL
LIN {X 0,Y 654.552,Z 777.697,A -85,B 0,C 180,E1 5954.922,E2 5954.922} C_VEL
LIN {X 0,Y 655.536,Z 747.983,A -85,B 0,C 180,E1 5956.61,E2 5956.61} C_VEL
LIN {X 0,Y 656.462,Z 714.344,A -85,B 0,C 180,E1 5957.893,E2 5957.893} C_VEL
LIN {X 0,Y 657.2,Z 678.728,A -85,B 0,C 180,E1 5958.698,E2 5958.698} C_VEL
LIN {X 0,Y 657.165,Z 620.66,A -85,B 0,C 180,E1 5959.499,E2 5959.499} C_VEL
LIN {X 0,Y 651.553,Z 603.959,A -85,B 0,C 180,E1 5959.952,E2 5959.952} C_VEL
LIN {X 0,Y 649.041,Z 599.629,A -85,B 0,C 180,E1 5960.355,E2 5960.355} C_VEL
LIN {X 0,Y 645.923,Z 598.648,A -85,B 0,C 180,E1 5961.155,E2 5961.155} C_VEL
LIN {X 0,Y 642.965,Z 601.31,A -85,B 0,C 180,E1 5962.928,E2 5962.928} C_VEL
LIN {X 0,Y 642.937,Z 601.31,A -85,B 0,C 180,E1 5968.117,E2 5968.117} C_VEL
LIN {X 0,Y 642.913,Z 601.31,A -85,B 0,C 180,E1 5972.818,E2 5972.818} C_VEL
LIN {X 0,Y 642.841,Z 601.31,A -85,B 0,C 180,E1 5977.787,E2 5977.787} C_VEL
LIN {X 0,Y 642.872,Z 601.31,A -85,B 0,C 180,E1 5983.109,E2 5983.109} C_VEL
LIN {X 0,Y 642.762,Z 601.31,A -85,B 0,C 180,E1 5988.957,E2 5988.957} C_VEL
LIN {X 0,Y 642.843,Z 601.357,A -85,B 0,C 180,E1 5994.566,E2 5994.566} C_VEL
LIN {X 0,Y 651.701,Z 624.734,A -85,B 0,C 180,E1 5995.172,E2 5995.172} C_VEL
LIN {X 0,Y 660.733,Z 643.14,A -85,B 0,C 180,E1 5995.719,E2 5995.719} C_VEL
LIN {X 0,Y 660.141,Z 712.081,A -85,B 0,C 180,E1 5996.612,E2 5996.612} C_VEL
LIN {X 0,Y 658.55,Z 757.265,A -85,B 0,C 180,E1 5997.724,E2 5997.724} C_VEL
LIN {X 0,Y 656.674,Z 793.905,A -85,B 0,C 180,E1 5999.102,E2 5999.102} C_VEL
LIN {X 0,Y 653.787,Z 835.971,A -85,B 0,C 180,E1 6001.309,E2 6001.309} C_VEL
LIN {X 0,Y 650.867,Z 873.889,A -85,B 0,C 180,E1 6003.938,E2 6003.938} C_VEL
LIN {X 0,Y 648.3,Z 907.601,A -85,B 0,C 180,E1 6006.94,E2 6006.94} C_VEL
LIN {X 0,Y 646.304,Z 936.501,A -85,B 0,C 180,E1 6010.207,E2 6010.207} C_VEL
LIN {X 0,Y 644.963,Z 961.543,A -85,B 0,C 180,E1 6013.855,E2 6013.855} C_VEL
LIN {X 0,Y 644.098,Z 981.627,A -85,B 0,C 180,E1 6017.781,E2 6017.781} C_VEL
LIN {X 0,Y 643.798,Z 994.314,A -85,B 0,C 180,E1 6021.229,E2 6021.229} C_VEL
LIN {X 0,Y 643.617,Z 1003.672,A -85,B 0,C 180,E1 6025.277,E2 6025.277} C_VEL
LIN {X 0,Y 643.65,Z 1007.168,A -85,B 0,C 180,E1 6028.655,E2 6028.655} C_VEL
LIN {X 0,Y 643.64,Z 1006.213,A -85,B 0,C 180,E1 6032.702,E2 6032.702} C_VEL
LIN {X 0,Y 643.688,Z 1001.189,A -85,B 0,C 180,E1 6036.084,E2 6036.084} C_VEL
LIN {X 0,Y 643.833,Z 989.706,A -85,B 0,C 180,E1 6040.17,E2 6040.17} C_VEL
LIN {X 0,Y 644.341,Z 973.518,A -85,B 0,C 180,E1 6043.951,E2 6043.951} C_VEL
LIN {X 0,Y 645.303,Z 952.349,A -85,B 0,C 180,E1 6047.6,E2 6047.6} C_VEL
LIN {X 0,Y 647.161,Z 924.239,A -85,B 0,C 180,E1 6051.283,E2 6051.283} C_VEL
LIN {X 0,Y 649.633,Z 890.126,A -85,B 0,C 180,E1 6054.716,E2 6054.716} C_VEL
LIN {X 0,Y 652.538,Z 851.905,A -85,B 0,C 180,E1 6057.676,E2 6057.676} C_VEL
LIN {X 0,Y 655.465,Z 810.999,A -85,B 0,C 180,E1 6060.081,E2 6060.081} C_VEL
LIN {X 0,Y 657.977,Z 771.034,A -85,B 0,C 180,E1 6061.815,E2 6061.815} C_VEL
LIN {X 0,Y 659.869,Z 727.065,A -85,B 0,C 180,E1 6063.112,E2 6063.112} C_VEL
LIN {X 0,Y 660.949,Z 680.24,A -85,B 0,C 180,E1 6063.934,E2 6063.934} C_VEL
LIN {X 0,Y 660.711,Z 640.032,A -85,B 0,C 180,E1 6064.44,E2 6064.44} C_VEL
LIN {X 0,Y 643.021,Z 602.568,A -85,B 0,C 180,E1 6065.794,E2 6065.794} C_VEL
LIN {X 0,Y 642.87,Z 601.31,A -85,B 0,C 180,E1 6065.92,E2 6065.92} C_VEL
LIN {X 0,Y 642.823,Z 601.31,A -85,B 0,C 180,E1 6071.304,E2 6071.304} C_VEL
LIN {X 0,Y 642.765,Z 601.31,A -85,B 0,C 180,E1 6076.956,E2 6076.956} C_VEL
LIN {X 0,Y 642.749,Z 601.31,A -85,B 0,C 180,E1 6082.206,E2 6082.206} C_VEL
LIN {X 0,Y 642.818,Z 601.31,A -85,B 0,C 180,E1 6087.176,E2 6087.176} C_VEL
LIN {X 0,Y 642.952,Z 601.31,A -85,B 0,C 180,E1 6091.884,E2 6091.884} C_VEL
LIN {X 0,Y 643.068,Z 601.31,A -85,B 0,C 180,E1 6096.778,E2 6096.778} C_VEL
LIN {X 0,Y 643.105,Z 601.31,A -85,B 0,C 180,E1 6102.166,E2 6102.166} C_VEL
LIN {X 0,Y 643.141,Z 601.31,A -85,B 0,C 180,E1 6107.759,E2 6107.759} C_VEL
LIN {X 0,Y 643.353,Z 601.31,A -85,B 0,C 180,E1 6113.237,E2 6113.237} C_VEL
LIN {X 0,Y 643.398,Z 601.31,A -85,B 0,C 180,E1 6118.649,E2 6118.649} C_VEL
LIN {X 0,Y 643.394,Z 601.31,A -85,B 0,C 180,E1 6122.697,E2 6122.697} C_VEL
LIN {X 0,Y 643.242,Z 601.31,A -85,B 0,C 180,E1 6126.761,E2 6126.761} C_VEL
LIN {X 0,Y 643.218,Z 601.31,A -85,B 0,C 180,E1 6132.236,E2 6132.236} C_VEL
LIN {X 0,Y 643.132,Z 601.31,A -85,B 0,C 180,E1 6137.829,E2 6137.829} C_VEL
LIN {X 0,Y 643.04,Z 601.31,A -85,B 0,C 180,E1 6143.216,E2 6143.216} C_VEL
LIN {X 0,Y 642.938,Z 601.31,A -85,B 0,C 180,E1 6148.113,E2 6148.113} C_VEL
LIN {X 0,Y 642.88,Z 601.31,A -85,B 0,C 180,E1 6152.816,E2 6152.816} C_VEL
LIN {X 0,Y 642.805,Z 601.31,A -85,B 0,C 180,E1 6157.785,E2 6157.785} C_VEL
LIN {X 0,Y 642.888,Z 601.31,A -85,B 0,C 180,E1 6163.103,E2 6163.103} C_VEL
LIN {X 0,Y 642.787,Z 601.31,A -85,B 0,C 180,E1 6168.949,E2 6168.949} C_VEL
LIN {X 0,Y 642.761,Z 601.31,A -85,B 0,C 180,E1 6173.886,E2 6173.886} C_VEL
LIN {X 0,Y 642.863,Z 601.31,A -85,B 0,C 180,E1 6178.762,E2 6178.762} C_VEL
LIN {X 0,Y 643.163,Z 601.979,A -85,B 0,C 180,E1 6183.095,E2 6183.095} C_VEL
LIN {X 0,Y 653.418,Z 634.783,A -85,B 0,C 180,E1 6184.047,E2 6184.047} C_VEL
LIN {X 0,Y 652.192,Z 672.743,A -85,B 0,C 180,E1 6185.151,E2 6185.151} C_VEL
LIN {X 0,Y 650.579,Z 708.74,A -85,B 0,C 180,E1 6186.727,E2 6186.727} C_VEL
LIN {X 0,Y 648.721,Z 743.343,A -85,B 0,C 180,E1 6188.833,E2 6188.833} C_VEL
LIN {X 0,Y 646.816,Z 774.316,A -85,B 0,C 180,E1 6191.405,E2 6191.405} C_VEL
LIN {X 0,Y 645.406,Z 801.191,A -85,B 0,C 180,E1 6194.335,E2 6194.335} C_VEL
LIN {X 0,Y 644.448,Z 822.428,A -85,B 0,C 180,E1 6197.429,E2 6197.429} C_VEL
LIN {X 0,Y 643.857,Z 839.617,A -85,B 0,C 180,E1 6200.917,E2 6200.917} C_VEL
LIN {X 0,Y 643.712,Z 849.567,A -85,B 0,C 180,E1 6203.916,E2 6203.916} C_VEL
LIN {X 0,Y 643.631,Z 855.939,A -85,B 0,C 180,E1 6207.298,E2 6207.298} C_VEL
LIN {X 0,Y 643.58,Z 857.409,A -85,B 0,C 180,E1 6209.996,E2 6209.996} C_VEL
LIN {X 0,Y 643.629,Z 855.829,A -85,B 0,C 180,E1 6212.695,E2 6212.695} C_VEL
LIN {X 0,Y 643.762,Z 849.345,A -85,B 0,C 180,E1 6216.076,E2 6216.076} C_VEL
LIN {X 0,Y 643.938,Z 837.628,A -85,B 0,C 180,E1 6219.477,E2 6219.477} C_VEL
LIN {X 0,Y 644.535,Z 820.859,A -85,B 0,C 180,E1 6222.753,E2 6222.753} C_VEL
LIN {X 0,Y 645.558,Z 797.563,A -85,B 0,C 180,E1 6226.013,E2 6226.013} C_VEL
LIN {X 0,Y 647.167,Z 769.473,A -85,B 0,C 180,E1 6228.966,E2 6228.966} C_VEL
LIN {X 0,Y 648.966,Z 738.711,A -85,B 0,C 180,E1 6231.397,E2 6231.397} C_VEL
LIN {X 0,Y 650.921,Z 702.785,A -85,B 0,C 180,E1 6233.489,E2 6233.489} C_VEL
LIN {X 0,Y 652.534,Z 664,A -85,B 0,C 180,E1 6235.063,E2 6235.063} C_VEL
LIN {X 0,Y 652.882,Z 631.457,A -85,B 0,C 180,E1 6235.962,E2 6235.962} C_VEL
LIN {X 0,Y 642.916,Z 601.31,A -85,B 0,C 180,E1 6236.913,E2 6236.913} C_VEL
LIN {X 0,Y 642.87,Z 601.31,A -85,B 0,C 180,E1 6241.974,E2 6241.974} C_VEL
LIN {X 0,Y 642.775,Z 601.31,A -85,B 0,C 180,E1 6246.748,E2 6246.748} C_VEL
LIN {X 0,Y 642.84,Z 601.31,A -85,B 0,C 180,E1 6251.293,E2 6251.293} C_VEL
LIN {X 0,Y 642.769,Z 601.31,A -85,B 0,C 180,E1 6256.945,E2 6256.945} C_VEL
LIN {X 0,Y 642.744,Z 601.31,A -85,B 0,C 180,E1 6262.21,E2 6262.21} C_VEL
LIN {X 0,Y 642.857,Z 601.31,A -85,B 0,C 180,E1 6267.183,E2 6267.183} C_VEL
LIN {X 0,Y 642.946,Z 601.31,A -85,B 0,C 180,E1 6271.888,E2 6271.888} C_VEL
LIN {X 0,Y 643.035,Z 601.31,A -85,B 0,C 180,E1 6276.766,E2 6276.766} C_VEL
LIN {X 0,Y 642.936,Z 601.31,A -85,B 0,C 180,E1 6279.787,E2 6279.787} C_VEL
LIN {X 0,Y 650.088,Z 626.589,A -85,B 0,C 180,E1 6280.361,E2 6280.361} C_VEL
LIN {X 0,Y 649.315,Z 693.967,A -85,B 0,C 180,E1 6281.291,E2 6281.291} C_VEL
LIN {X 0,Y 648.53,Z 729.028,A -85,B 0,C 180,E1 6282.324,E2 6282.324} C_VEL
LIN {X 0,Y 647.332,Z 760.747,A -85,B 0,C 180,E1 6283.805,E2 6283.805} C_VEL
LIN {X 0,Y 646.241,Z 789.699,A -85,B 0,C 180,E1 6285.753,E2 6285.753} C_VEL
LIN {X 0,Y 645.217,Z 815.077,A -85,B 0,C 180,E1 6288.147,E2 6288.147} C_VEL
LIN {X 0,Y 644.563,Z 835.205,A -85,B 0,C 180,E1 6290.84,E2 6290.84} C_VEL
LIN {X 0,Y 644.194,Z 849.107,A -85,B 0,C 180,E1 6293.588,E2 6293.588} C_VEL
LIN {X 0,Y 644.035,Z 858.365,A -85,B 0,C 180,E1 6296.631,E2 6296.631} C_VEL
LIN {X 0,Y 643.948,Z 861.275,A -85,B 0,C 180,E1 6298.654,E2 6298.654} C_VEL
LIN {X 0,Y 643.966,Z 861.419,A -85,B 0,C 180,E1 6301.35,E2 6301.35} C_VEL
LIN {X 0,Y 644.121,Z 857.217,A -85,B 0,C 180,E1 6304.048,E2 6304.048} C_VEL
LIN {X 0,Y 644.403,Z 846.82,A -85,B 0,C 180,E1 6307.091,E2 6307.091} C_VEL
LIN {X 0,Y 644.92,Z 831.76,A -85,B 0,C 180,E1 6309.807,E2 6309.807} C_VEL
LIN {X 0,Y 645.619,Z 811.454,A -85,B 0,C 180,E1 6312.319,E2 6312.319} C_VEL
LIN {X 0,Y 646.681,Z 785.629,A -85,B 0,C 180,E1 6314.587,E2 6314.587} C_VEL
LIN {X 0,Y 647.73,Z 755.641,A -85,B 0,C 180,E1 6316.458,E2 6316.458} C_VEL
LIN {X 0,Y 648.811,Z 721.783,A -85,B 0,C 180,E1 6317.891,E2 6317.891} C_VEL
LIN {X 0,Y 649.68,Z 684.979,A -85,B 0,C 180,E1 6318.834,E2 6318.834} C_VEL
LIN {X 0,Y 649.832,Z 622.286,A -85,B 0,C 180,E1 6319.751,E2 6319.751} C_VEL
LIN {X 0,Y 643.133,Z 601.31,A -85,B 0,C 180,E1 6320.385,E2 6320.385} C_VEL
LIN {X 0,Y 642.965,Z 601.31,A -85,B 0,C 180,E1 6322.928,E2 6322.928} C_VEL
LIN {X 0,Y 640.465,Z 601.31,A -85,B 0,C 180,E1 6324.08,E2 6324.08} C_VEL
LIN {X 0,Y 635.074,Z 601.31,A -85,B 0,C 180,E1 6325.801,E2 6325.801} C_VEL
LIN {X 0,Y 634.973,Z 601.31,A -85,B 0,C 180,E1 6325.999,E2 6325.999} C_VEL
LIN {X 0,Y 634.951,Z 601.31,A -85,B 0,C 180,E1 6330.794,E2 6330.794} C_VEL
LIN {X 0,Y 634.932,Z 601.31,A -85,B 0,C 180,E1 6335.776,E2 6335.776} C_VEL
LIN {X 0,Y 634.886,Z 601.31,A -85,B 0,C 180,E1 6340.214,E2 6340.214} C_VEL
LIN {X 0,Y 634.874,Z 601.31,A -85,B 0,C 180,E1 6345.714,E2 6345.714} C_VEL
LIN {X 0,Y 634.829,Z 601.31,A -85,B 0,C 180,E1 6351.647,E2 6351.647} C_VEL
LIN {X 0,Y 634.947,Z 602.12,A -85,B 0,C 180,E1 6354.255,E2 6354.255} C_VEL
LIN {X 0,Y 645.658,Z 629.417,A -85,B 0,C 180,E1 6354.995,E2 6354.995} C_VEL
LIN {X 0,Y 653.471,Z 645.047,A -85,B 0,C 180,E1 6355.468,E2 6355.468} C_VEL
LIN {X 0,Y 652.85,Z 712.168,A -85,B 0,C 180,E1 6356.35,E2 6356.35} C_VEL
LIN {X 0,Y 651.195,Z 757.347,A -85,B 0,C 180,E1 6357.475,E2 6357.475} C_VEL
LIN {X 0,Y 649.18,Z 799.679,A -85,B 0,C 180,E1 6359.054,E2 6359.054} C_VEL
LIN {X 0,Y 646.709,Z 834.902,A -85,B 0,C 180,E1 6360.898,E2 6360.898} C_VEL
LIN {X 0,Y 643.721,Z 871.582,A -85,B 0,C 180,E1 6363.438,E2 6363.438} C_VEL
LIN {X 0,Y 640.994,Z 905.637,A -85,B 0,C 180,E1 6366.455,E2 6366.455} C_VEL
LIN {X 0,Y 638.671,Z 935.88,A -85,B 0,C 180,E1 6369.877,E2 6369.877} C_VEL
LIN {X 0,Y 637.182,Z 961.369,A -85,B 0,C 180,E1 6373.625,E2 6373.625} C_VEL
LIN {X 0,Y 636.302,Z 980.881,A -85,B 0,C 180,E1 6377.459,E2 6377.459} C_VEL
LIN {X 0,Y 635.91,Z 994.314,A -85,B 0,C 180,E1 6381.119,E2 6381.119} C_VEL
LIN {X 0,Y 635.74,Z 1003.672,A -85,B 0,C 180,E1 6385.219,E2 6385.219} C_VEL
LIN {X 0,Y 635.76,Z 1007.168,A -85,B 0,C 180,E1 6388.638,E2 6388.638} C_VEL
LIN {X 0,Y 635.755,Z 1006.213,A -85,B 0,C 180,E1 6392.736,E2 6392.736} C_VEL
LIN {X 0,Y 635.793,Z 1001.19,A -85,B 0,C 180,E1 6396.16,E2 6396.16} C_VEL
LIN {X 0,Y 635.961,Z 989.707,A -85,B 0,C 180,E1 6400.297,E2 6400.297} C_VEL
LIN {X 0,Y 636.537,Z 973.517,A -85,B 0,C 180,E1 6404.126,E2 6404.126} C_VEL
LIN {X 0,Y 637.608,Z 952.347,A -85,B 0,C 180,E1 6407.82,E2 6407.82} C_VEL
LIN {X 0,Y 639.601,Z 924.237,A -85,B 0,C 180,E1 6411.547,E2 6411.547} C_VEL
LIN {X 0,Y 642.24,Z 890.554,A -85,B 0,C 180,E1 6414.981,E2 6414.981} C_VEL
LIN {X 0,Y 645.38,Z 851.902,A -85,B 0,C 180,E1 6418.01,E2 6418.01} C_VEL
LIN {X 0,Y 648.376,Z 811.933,A -85,B 0,C 180,E1 6420.378,E2 6420.378} C_VEL
LIN {X 0,Y 650.814,Z 770.401,A -85,B 0,C 180,E1 6422.14,E2 6422.14} C_VEL
LIN {X 0,Y 652.823,Z 727.218,A -85,B 0,C 180,E1 6423.426,E2 6423.426} C_VEL
LIN {X 0,Y 654.001,Z 679.91,A -85,B 0,C 180,E1 6424.265,E2 6424.265} C_VEL
LIN {X 0,Y 653.754,Z 642.426,A -85,B 0,C 180,E1 6424.75,E2 6424.75} C_VEL
LIN {X 0,Y 635.137,Z 603.12,A -85,B 0,C 180,E1 6426.206,E2 6426.206} C_VEL
LIN {X 0,Y 634.925,Z 601.31,A -85,B 0,C 180,E1 6426.3,E2 6426.3} C_VEL
LIN {X 0,Y 634.862,Z 601.31,A -85,B 0,C 180,E1 6432.291,E2 6432.291} C_VEL
LIN {X 0,Y 634.801,Z 601.31,A -85,B 0,C 180,E1 6437.732,E2 6437.732} C_VEL
LIN {X 0,Y 634.861,Z 601.31,A -85,B 0,C 180,E1 6443.375,E2 6443.375} C_VEL
LIN {X 0,Y 634.92,Z 601.31,A -85,B 0,C 180,E1 6449.225,E2 6449.225} C_VEL
LIN {X 0,Y 635.094,Z 601.31,A -85,B 0,C 180,E1 6454.572,E2 6454.572} C_VEL
LIN {X 0,Y 635.115,Z 601.31,A -85,B 0,C 180,E1 6459.034,E2 6459.034} C_VEL
LIN {X 0,Y 635.183,Z 601.31,A -85,B 0,C 180,E1 6463.368,E2 6463.368} C_VEL
LIN {X 0,Y 635.278,Z 601.31,A -85,B 0,C 180,E1 6469.001,E2 6469.001} C_VEL
LIN {X 0,Y 635.419,Z 601.31,A -85,B 0,C 180,E1 6474.526,E2 6474.526} C_VEL
LIN {X 0,Y 635.497,Z 601.31,A -85,B 0,C 180,E1 6478.632,E2 6478.632} C_VEL
LIN {X 0,Y 635.503,Z 601.31,A -85,B 0,C 180,E1 6482.731,E2 6482.731} C_VEL
LIN {X 0,Y 635.333,Z 601.31,A -85,B 0,C 180,E1 6486.845,E2 6486.845} C_VEL
LIN {X 0,Y 635.296,Z 601.31,A -85,B 0,C 180,E1 6492.391,E2 6492.391} C_VEL
LIN {X 0,Y 635.208,Z 601.31,A -85,B 0,C 180,E1 6498.059,E2 6498.059} C_VEL
LIN {X 0,Y 635.108,Z 601.31,A -85,B 0,C 180,E1 6502.433,E2 6502.433} C_VEL
LIN {X 0,Y 635.052,Z 601.31,A -85,B 0,C 180,E1 6508.01,E2 6508.01} C_VEL
LIN {X 0,Y 634.923,Z 601.31,A -85,B 0,C 180,E1 6513.351,E2 6513.351} C_VEL
LIN {X 0,Y 634.896,Z 601.31,A -85,B 0,C 180,E1 6518.341,E2 6518.341} C_VEL
LIN {X 0,Y 634.921,Z 601.31,A -85,B 0,C 180,E1 6524.275,E2 6524.275} C_VEL
LIN {X 0,Y 634.839,Z 601.31,A -85,B 0,C 180,E1 6529.873,E2 6529.873} C_VEL
LIN {X 0,Y 634.867,Z 601.31,A -85,B 0,C 180,E1 6535.05,E2 6535.05} C_VEL
LIN {X 0,Y 634.955,Z 601.31,A -85,B 0,C 180,E1 6539.921,E2 6539.921} C_VEL
LIN {X 0,Y 635.191,Z 601.31,A -85,B 0,C 180,E1 6542.79,E2 6542.79} C_VEL
LIN {X 0,Y 646.012,Z 636.283,A -85,B 0,C 180,E1 6543.827,E2 6543.827} C_VEL
LIN {X 0,Y 644.721,Z 674.523,A -85,B 0,C 180,E1 6544.97,E2 6544.97} C_VEL
LIN {X 0,Y 643.068,Z 710.958,A -85,B 0,C 180,E1 6546.591,E2 6546.591} C_VEL
LIN {X 0,Y 641.13,Z 744.999,A -85,B 0,C 180,E1 6548.698,E2 6548.698} C_VEL
LIN {X 0,Y 639.195,Z 775.389,A -85,B 0,C 180,E1 6551.253,E2 6551.253} C_VEL
LIN {X 0,Y 637.591,Z 802.582,A -85,B 0,C 180,E1 6554.314,E2 6554.314} C_VEL
LIN {X 0,Y 636.567,Z 824.389,A -85,B 0,C 180,E1 6557.626,E2 6557.626} C_VEL
LIN {X 0,Y 635.982,Z 840.599,A -85,B 0,C 180,E1 6561.048,E2 6561.048} C_VEL
LIN {X 0,Y 635.82,Z 851.323,A -85,B 0,C 180,E1 6564.526,E2 6564.526} C_VEL
LIN {X 0,Y 635.743,Z 855.934,A -85,B 0,C 180,E1 6567.264,E2 6567.264} C_VEL
LIN {X 0,Y 635.68,Z 857.402,A -85,B 0,C 180,E1 6569.996,E2 6569.996} C_VEL
LIN {X 0,Y 635.742,Z 855.826,A -85,B 0,C 180,E1 6572.728,E2 6572.728} C_VEL
LIN {X 0,Y 635.869,Z 849.341,A -85,B 0,C 180,E1 6576.152,E2 6576.152} C_VEL
LIN {X 0,Y 636.069,Z 837.624,A -85,B 0,C 180,E1 6579.595,E2 6579.595} C_VEL
LIN {X 0,Y 636.719,Z 821.202,A -85,B 0,C 180,E1 6582.855,E2 6582.855} C_VEL
LIN {X 0,Y 637.738,Z 799.279,A -85,B 0,C 180,E1 6586.003,E2 6586.003} C_VEL
LIN {X 0,Y 639.452,Z 771.806,A -85,B 0,C 180,E1 6589.002,E2 6589.002} C_VEL
LIN {X 0,Y 641.282,Z 742.373,A -85,B 0,C 180,E1 6591.396,E2 6591.396} C_VEL
LIN {X 0,Y 643.107,Z 709.232,A -85,B 0,C 180,E1 6593.411,E2 6593.411} C_VEL
LIN {X 0,Y 644.856,Z 672.495,A -85,B 0,C 180,E1 6595.016,E2 6595.016} C_VEL
LIN {X 0,Y 645.572,Z 633.644,A -85,B 0,C 180,E1 6596.164,E2 6596.164} C_VEL
LIN {X 0,Y 635.01,Z 601.31,A -85,B 0,C 180,E1 6597.166,E2 6597.166} C_VEL
LIN {X 0,Y 634.965,Z 601.31,A -85,B 0,C 180,E1 6601.663,E2 6601.663} C_VEL
LIN {X 0,Y 634.887,Z 601.31,A -85,B 0,C 180,E1 6606.625,E2 6606.625} C_VEL
LIN {X 0,Y 634.908,Z 601.31,A -85,B 0,C 180,E1 6612.301,E2 6612.301} C_VEL
LIN {X 0,Y 634.793,Z 601.31,A -85,B 0,C 180,E1 6617.721,E2 6617.721} C_VEL
LIN {X 0,Y 634.85,Z 601.31,A -85,B 0,C 180,E1 6623.379,E2 6623.379} C_VEL
LIN {X 0,Y 634.927,Z 601.31,A -85,B 0,C 180,E1 6628.34,E2 6628.34} C_VEL
LIN {X 0,Y 635.066,Z 601.31,A -85,B 0,C 180,E1 6633.051,E2 6633.051} C_VEL
LIN {X 0,Y 635.017,Z 601.31,A -85,B 0,C 180,E1 6638.514,E2 6638.514} C_VEL
LIN {X 0,Y 635.024,Z 601.31,A -85,B 0,C 180,E1 6639.508,E2 6639.508} C_VEL
LIN {X 0,Y 642.701,Z 629.237,A -85,B 0,C 180,E1 6640.149,E2 6640.149} C_VEL
LIN {X 0,Y 641.841,Z 694.199,A -85,B 0,C 180,E1 6641.065,E2 6641.065} C_VEL
LIN {X 0,Y 641.006,Z 729.267,A -85,B 0,C 180,E1 6642.11,E2 6642.11} C_VEL
LIN {X 0,Y 639.715,Z 762.51,A -85,B 0,C 180,E1 6643.688,E2 6643.688} C_VEL
LIN {X 0,Y 638.535,Z 791.217,A -85,B 0,C 180,E1 6645.665,E2 6645.665} C_VEL
LIN {X 0,Y 637.496,Z 815.663,A -85,B 0,C 180,E1 6648.001,E2 6648.001} C_VEL
LIN {X 0,Y 636.776,Z 835.929,A -85,B 0,C 180,E1 6650.727,E2 6650.727} C_VEL
LIN {X 0,Y 636.382,Z 849.957,A -85,B 0,C 180,E1 6653.509,E2 6653.509} C_VEL
LIN {X 0,Y 636.225,Z 859.308,A -85,B 0,C 180,E1 6656.589,E2 6656.589} C_VEL
LIN {X 0,Y 636.114,Z 862.283,A -85,B 0,C 180,E1 6658.637,E2 6658.637} C_VEL
LIN {X 0,Y 636.169,Z 862.466,A -85,B 0,C 180,E1 6661.366,E2 6661.366} C_VEL
LIN {X 0,Y 636.334,Z 858.274,A -85,B 0,C 180,E1 6664.097,E2 6664.097} C_VEL
LIN {X 0,Y 636.646,Z 847.853,A -85,B 0,C 180,E1 6667.178,E2 6667.178} C_VEL
LIN {X 0,Y 637.193,Z 832.733,A -85,B 0,C 180,E1 6669.927,E2 6669.927} C_VEL
LIN {X 0,Y 637.929,Z 812.404,A -85,B 0,C 180,E1 6672.461,E2 6672.461} C_VEL
LIN {X 0,Y 639.074,Z 786.386,A -85,B 0,C 180,E1 6674.765,E2 6674.765} C_VEL
LIN {X 0,Y 640.188,Z 756.335,A -85,B 0,C 180,E1 6676.657,E2 6676.657} C_VEL
LIN {X 0,Y 641.336,Z 722.435,A -85,B 0,C 180,E1 6678.107,E2 6678.107} C_VEL
LIN {X 0,Y 642.261,Z 686.283,A -85,B 0,C 180,E1 6679.06,E2 6679.06} C_VEL
LIN {X 0,Y 642.78,Z 624.674,A -85,B 0,C 180,E1 6679.981,E2 6679.981} C_VEL
LIN {X 0,Y 635.17,Z 601.31,A -85,B 0,C 180,E1 6680.737,E2 6680.737} C_VEL
LIN {X 0,Y 634.973,Z 601.31,A -85,B 0,C 180,E1 6685.999,E2 6685.999} C_VEL
LIN {X 0,Y 631.026,Z 601.31,A -85,B 0,C 180,E1 6687.538,E2 6687.538} C_VEL
LIN {X 0,Y 627.052,Z 601.31,A -85,B 0,C 180,E1 6689.095,E2 6689.095} C_VEL
LIN {X 0,Y 627.022,Z 601.31,A -85,B 0,C 180,E1 6694.76,E2 6694.76} C_VEL
LIN {X 0,Y 626.949,Z 601.31,A -85,B 0,C 180,E1 6699.348,E2 6699.348} C_VEL
LIN {X 0,Y 626.998,Z 601.31,A -85,B 0,C 180,E1 6704.483,E2 6704.483} C_VEL
LIN {X 0,Y 626.858,Z 601.31,A -85,B 0,C 180,E1 6709.265,E2 6709.265} C_VEL
LIN {X 0,Y 626.964,Z 601.31,A -85,B 0,C 180,E1 6713.877,E2 6713.877} C_VEL
LIN {X 0,Y 638.753,Z 632.492,A -85,B 0,C 180,E1 6714.762,E2 6714.762} C_VEL
LIN {X 0,Y 646.078,Z 646.285,A -85,B 0,C 180,E1 6715.201,E2 6715.201} C_VEL
LIN {X 0,Y 645.56,Z 712.402,A -85,B 0,C 180,E1 6716.085,E2 6716.085} C_VEL
LIN {X 0,Y 643.809,Z 757.856,A -85,B 0,C 180,E1 6717.232,E2 6717.232} C_VEL
LIN {X 0,Y 641.666,Z 800.821,A -85,B 0,C 180,E1 6718.867,E2 6718.867} C_VEL
LIN {X 0,Y 639.22,Z 839.639,A -85,B 0,C 180,E1 6720.867,E2 6720.867} C_VEL
LIN {X 0,Y 636.198,Z 875.304,A -85,B 0,C 180,E1 6723.408,E2 6723.408} C_VEL
LIN {X 0,Y 633.239,Z 909.115,A -85,B 0,C 180,E1 6726.521,E2 6726.521} C_VEL
LIN {X 0,Y 630.899,Z 937.73,A -85,B 0,C 180,E1 6729.872,E2 6729.872} C_VEL
LIN {X 0,Y 629.365,Z 962.123,A -85,B 0,C 180,E1 6733.543,E2 6733.543} C_VEL
LIN {X 0,Y 628.435,Z 981.625,A -85,B 0,C 180,E1 6737.471,E2 6737.471} C_VEL
LIN {X 0,Y 628.036,Z 994.438,A -85,B 0,C 180,E1 6741.051,E2 6741.051} C_VEL
LIN {X 0,Y 627.862,Z 1003.673,A -85,B 0,C 180,E1 6745.159,E2 6745.159} C_VEL
LIN {X 0,Y 627.856,Z 1007.167,A -85,B 0,C 180,E1 6748.621,E2 6748.621} C_VEL
LIN {X 0,Y 627.849,Z 1006.212,A -85,B 0,C 180,E1 6752.77,E2 6752.77} C_VEL
LIN {X 0,Y 627.88,Z 1001.19,A -85,B 0,C 180,E1 6756.238,E2 6756.238} C_VEL
LIN {X 0,Y 628.101,Z 989.707,A -85,B 0,C 180,E1 6760.428,E2 6760.428} C_VEL
LIN {X 0,Y 628.728,Z 973.516,A -85,B 0,C 180,E1 6764.305,E2 6764.305} C_VEL
LIN {X 0,Y 629.907,Z 952.345,A -85,B 0,C 180,E1 6768.045,E2 6768.045} C_VEL
LIN {X 0,Y 632.031,Z 924.236,A -85,B 0,C 180,E1 6771.818,E2 6771.818} C_VEL
LIN {X 0,Y 634.922,Z 890.021,A -85,B 0,C 180,E1 6775.339,E2 6775.339} C_VEL
LIN {X 0,Y 638.21,Z 851.896,A -85,B 0,C 180,E1 6778.353,E2 6778.353} C_VEL
LIN {X 0,Y 640.982,Z 813.146,A -85,B 0,C 180,E1 6780.601,E2 6780.601} C_VEL
LIN {X 0,Y 643.6,Z 772.132,A -85,B 0,C 180,E1 6782.385,E2 6782.385} C_VEL
LIN {X 0,Y 645.774,Z 727.845,A -85,B 0,C 180,E1 6783.736,E2 6783.736} C_VEL
LIN {X 0,Y 647.069,Z 680.787,A -85,B 0,C 180,E1 6784.586,E2 6784.586} C_VEL
LIN {X 0,Y 647.066,Z 645.348,A -85,B 0,C 180,E1 6785.045,E2 6785.045} C_VEL
LIN {X 0,Y 627.178,Z 602.861,A -85,B 0,C 180,E1 6786.644,E2 6786.644} C_VEL
LIN {X 0,Y 627.013,Z 601.31,A -85,B 0,C 180,E1 6786.761,E2 6786.761} C_VEL
LIN {X 0,Y 626.928,Z 601.31,A -85,B 0,C 180,E1 6792.593,E2 6792.593} C_VEL
LIN {X 0,Y 626.871,Z 601.31,A -85,B 0,C 180,E1 6797.416,E2 6797.416} C_VEL
LIN {X 0,Y 626.939,Z 601.31,A -85,B 0,C 180,E1 6802.903,E2 6802.903} C_VEL
LIN {X 0,Y 626.956,Z 601.31,A -85,B 0,C 180,E1 6807.886,E2 6807.886} C_VEL
LIN {X 0,Y 627.137,Z 601.31,A -85,B 0,C 180,E1 6813.382,E2 6813.382} C_VEL
LIN {X 0,Y 627.195,Z 601.31,A -85,B 0,C 180,E1 6818.757,E2 6818.757} C_VEL
LIN {X 0,Y 627.271,Z 601.31,A -85,B 0,C 180,E1 6823.152,E2 6823.152} C_VEL
LIN {X 0,Y 627.361,Z 601.31,A -85,B 0,C 180,E1 6828.86,E2 6828.86} C_VEL
LIN {X 0,Y 627.513,Z 601.31,A -85,B 0,C 180,E1 6834.457,E2 6834.457} C_VEL
LIN {X 0,Y 627.597,Z 601.31,A -85,B 0,C 180,E1 6838.615,E2 6838.615} C_VEL
LIN {X 0,Y 627.6,Z 601.31,A -85,B 0,C 180,E1 6842.765,E2 6842.765} C_VEL
LIN {X 0,Y 627.442,Z 601.31,A -85,B 0,C 180,E1 6848.04,E2 6848.04} C_VEL
LIN {X 0,Y 627.373,Z 601.31,A -85,B 0,C 180,E1 6852.55,E2 6852.55} C_VEL
LIN {X 0,Y 627.314,Z 601.31,A -85,B 0,C 180,E1 6856.843,E2 6856.843} C_VEL
LIN {X 0,Y 627.237,Z 601.31,A -85,B 0,C 180,E1 6861.238,E2 6861.238} C_VEL
LIN {X 0,Y 627.12,Z 601.31,A -85,B 0,C 180,E1 6866.615,E2 6866.615} C_VEL
LIN {X 0,Y 626.998,Z 601.31,A -85,B 0,C 180,E1 6872.234,E2 6872.234} C_VEL
LIN {X 0,Y 626.992,Z 601.31,A -85,B 0,C 180,E1 6877.157,E2 6877.157} C_VEL
LIN {X 0,Y 626.96,Z 601.31,A -85,B 0,C 180,E1 6882.572,E2 6882.572} C_VEL
LIN {X 0,Y 626.889,Z 601.31,A -85,B 0,C 180,E1 6887.403,E2 6887.403} C_VEL
LIN {X 0,Y 626.914,Z 601.31,A -85,B 0,C 180,E1 6892.881,E2 6892.881} C_VEL
LIN {X 0,Y 626.983,Z 601.31,A -85,B 0,C 180,E1 6897.877,E2 6897.877} C_VEL
LIN {X 0,Y 627.24,Z 601.597,A -85,B 0,C 180,E1 6902.509,E2 6902.509} C_VEL
LIN {X 0,Y 638.598,Z 637.544,A -85,B 0,C 180,E1 6903.604,E2 6903.604} C_VEL
LIN {X 0,Y 637.277,Z 675.52,A -85,B 0,C 180,E1 6904.751,E2 6904.751} C_VEL
LIN {X 0,Y 635.565,Z 711.849,A -85,B 0,C 180,E1 6906.392,E2 6906.392} C_VEL
LIN {X 0,Y 633.5,Z 746.832,A -85,B 0,C 180,E1 6908.583,E2 6908.583} C_VEL
LIN {X 0,Y 631.479,Z 777.986,A -85,B 0,C 180,E1 6911.248,E2 6911.248} C_VEL
LIN {X 0,Y 629.902,Z 803.157,A -85,B 0,C 180,E1 6914.143,E2 6914.143} C_VEL
LIN {X 0,Y 628.74,Z 824.381,A -85,B 0,C 180,E1 6917.47,E2 6917.47} C_VEL
LIN {X 0,Y 628.101,Z 840.581,A -85,B 0,C 180,E1 6920.933,E2 6920.933} C_VEL
LIN {X 0,Y 627.919,Z 851.325,A -85,B 0,C 180,E1 6924.457,E2 6924.457} C_VEL
LIN {X 0,Y 627.84,Z 855.929,A -85,B 0,C 180,E1 6927.23,E2 6927.23} C_VEL
LIN {X 0,Y 627.78,Z 857.396,A -85,B 0,C 180,E1 6929.996,E2 6929.996} C_VEL
LIN {X 0,Y 627.84,Z 855.822,A -85,B 0,C 180,E1 6932.763,E2 6932.763} C_VEL
LIN {X 0,Y 627.965,Z 849.337,A -85,B 0,C 180,E1 6936.23,E2 6936.23} C_VEL
LIN {X 0,Y 628.204,Z 837.62,A -85,B 0,C 180,E1 6939.716,E2 6939.716} C_VEL
LIN {X 0,Y 628.932,Z 819.998,A -85,B 0,C 180,E1 6943.227,E2 6943.227} C_VEL
LIN {X 0,Y 630.249,Z 797.418,A -85,B 0,C 180,E1 6946.497,E2 6946.497} C_VEL
LIN {X 0,Y 631.938,Z 771.345,A -85,B 0,C 180,E1 6949.298,E2 6949.298} C_VEL
LIN {X 0,Y 633.87,Z 740.945,A -85,B 0,C 180,E1 6951.742,E2 6951.742} C_VEL
LIN {X 0,Y 635.839,Z 706.55,A -85,B 0,C 180,E1 6953.798,E2 6953.798} C_VEL
LIN {X 0,Y 637.623,Z 667.355,A -85,B 0,C 180,E1 6955.454,E2 6955.454} C_VEL
LIN {X 0,Y 637.884,Z 634.853,A -85,B 0,C 180,E1 6956.4,E2 6956.4} C_VEL
LIN {X 0,Y 627.119,Z 601.31,A -85,B 0,C 180,E1 6957.451,E2 6957.451} C_VEL
LIN {X 0,Y 627.01,Z 601.31,A -85,B 0,C 180,E1 6962.265,E2 6962.265} C_VEL
LIN {X 0,Y 626.963,Z 601.31,A -85,B 0,C 180,E1 6967.165,E2 6967.165} C_VEL
LIN {X 0,Y 626.979,Z 601.31,A -85,B 0,C 180,E1 6972.579,E2 6972.579} C_VEL
LIN {X 0,Y 626.867,Z 601.31,A -85,B 0,C 180,E1 6977.42,E2 6977.42} C_VEL
LIN {X 0,Y 626.931,Z 601.31,A -85,B 0,C 180,E1 6982.892,E2 6982.892} C_VEL
LIN {X 0,Y 626.969,Z 601.31,A -85,B 0,C 180,E1 6987.891,E2 6987.891} C_VEL
LIN {X 0,Y 627.151,Z 601.31,A -85,B 0,C 180,E1 6993.362,E2 6993.362} C_VEL
LIN {X 0,Y 627.1,Z 601.31,A -85,B 0,C 180,E1 6998.757,E2 6998.757} C_VEL
LIN {X 0,Y 627.124,Z 601.31,A -85,B 0,C 180,E1 6999.215,E2 6999.215} C_VEL
LIN {X 0,Y 635.299,Z 629.754,A -85,B 0,C 180,E1 6999.908,E2 6999.908} C_VEL
LIN {X 0,Y 634.389,Z 694.03,A -85,B 0,C 180,E1 7000.828,E2 7000.828} C_VEL
LIN {X 0,Y 633.466,Z 729.409,A -85,B 0,C 180,E1 7001.889,E2 7001.889} C_VEL
LIN {X 0,Y 632.112,Z 762.78,A -85,B 0,C 180,E1 7003.487,E2 7003.487} C_VEL
LIN {X 0,Y 630.874,Z 791.642,A -85,B 0,C 180,E1 7005.487,E2 7005.487} C_VEL
LIN {X 0,Y 629.762,Z 816.247,A -85,B 0,C 180,E1 7007.851,E2 7007.851} C_VEL
LIN {X 0,Y 629.02,Z 836.12,A -85,B 0,C 180,E1 7010.529,E2 7010.529} C_VEL
LIN {X 0,Y 628.578,Z 850.785,A -85,B 0,C 180,E1 7013.428,E2 7013.428} C_VEL
LIN {X 0,Y 628.391,Z 860.253,A -85,B 0,C 180,E1 7016.547,E2 7016.547} C_VEL
LIN {X 0,Y 628.293,Z 863.274,A -85,B 0,C 180,E1 7018.62,E2 7018.62} C_VEL
LIN {X 0,Y 628.348,Z 863.514,A -85,B 0,C 180,E1 7021.383,E2 7021.383} C_VEL
LIN {X 0,Y 628.523,Z 859.345,A -85,B 0,C 180,E1 7024.148,E2 7024.148} C_VEL
LIN {X 0,Y 628.839,Z 850.405,A -85,B 0,C 180,E1 7026.92,E2 7026.92} C_VEL
LIN {X 0,Y 629.446,Z 834.843,A -85,B 0,C 180,E1 7029.875,E2 7029.875} C_VEL
LIN {X 0,Y 630.255,Z 814.409,A -85,B 0,C 180,E1 7032.495,E2 7032.495} C_VEL
LIN {X 0,Y 631.412,Z 789.553,A -85,B 0,C 180,E1 7034.77,E2 7034.77} C_VEL
LIN {X 0,Y 632.558,Z 759.945,A -85,B 0,C 180,E1 7036.703,E2 7036.703} C_VEL
LIN {X 0,Y 633.763,Z 725.845,A -85,B 0,C 180,E1 7038.236,E2 7038.236} C_VEL
LIN {X 0,Y 634.79,Z 689.968,A -85,B 0,C 180,E1 7039.246,E2 7039.246} C_VEL
LIN {X 0,Y 635.401,Z 626.011,A -85,B 0,C 180,E1 7040.259,E2 7040.259} C_VEL
LIN {X 0,Y 627.21,Z 601.31,A -85,B 0,C 180,E1 7041.035,E2 7041.035} C_VEL
LIN {X 0,Y 627.097,Z 601.31,A -85,B 0,C 180,E1 7046.628,E2 7046.628} C_VEL
LIN {X 0,Y 627.052,Z 601.31,A -85,B 0,C 180,E1 7049.095,E2 7049.095} C_VEL
LIN {X 0,Y 625.748,Z 601.31,A -85,B 0,C 180,E1 7049.887,E2 7049.887} C_VEL
LIN {X 0,Y 619.134,Z 601.31,A -85,B 0,C 180,E1 7052.039,E2 7052.039} C_VEL
LIN {X 0,Y 619.057,Z 601.31,A -85,B 0,C 180,E1 7052.243,E2 7052.243} C_VEL
LIN {X 0,Y 619.034,Z 601.31,A -85,B 0,C 180,E1 7057.721,E2 7057.721} C_VEL
LIN {X 0,Y 619.084,Z 601.31,A -85,B 0,C 180,E1 7063.25,E2 7063.25} C_VEL
LIN {X 0,Y 618.941,Z 601.31,A -85,B 0,C 180,E1 7068.631,E2 7068.631} C_VEL
LIN {X 0,Y 619.077,Z 601.966,A -85,B 0,C 180,E1 7073.557,E2 7073.557} C_VEL
LIN {X 0,Y 632.607,Z 636.962,A -85,B 0,C 180,E1 7074.565,E2 7074.565} C_VEL
LIN {X 0,Y 638.922,Z 649.393,A -85,B 0,C 180,E1 7074.962,E2 7074.962} C_VEL
LIN {X 0,Y 638.254,Z 713.073,A -85,B 0,C 180,E1 7075.823,E2 7075.823} C_VEL
LIN {X 0,Y 636.364,Z 759.851,A -85,B 0,C 180,E1 7077.029,E2 7077.029} C_VEL
LIN {X 0,Y 633.936,Z 804.833,A -85,B 0,C 180,E1 7078.802,E2 7078.802} C_VEL
LIN {X 0,Y 631.144,Z 846.661,A -85,B 0,C 180,E1 7081.077,E2 7081.077} C_VEL
LIN {X 0,Y 628.642,Z 878.512,A -85,B 0,C 180,E1 7083.337,E2 7083.337} C_VEL
LIN {X 0,Y 625.446,Z 913.029,A -85,B 0,C 180,E1 7086.633,E2 7086.633} C_VEL
LIN {X 0,Y 622.958,Z 942.57,A -85,B 0,C 180,E1 7090.281,E2 7090.281} C_VEL
LIN {X 0,Y 621.437,Z 965.549,A -85,B 0,C 180,E1 7093.962,E2 7093.962} C_VEL
LIN {X 0,Y 620.505,Z 983.86,A -85,B 0,C 180,E1 7097.851,E2 7097.851} C_VEL
LIN {X 0,Y 620.095,Z 996.172,A -85,B 0,C 180,E1 7101.573,E2 7101.573} C_VEL
LIN {X 0,Y 619.991,Z 1003.673,A -85,B 0,C 180,E1 7105.097,E2 7105.097} C_VEL
LIN {X 0,Y 619.966,Z 1007.167,A -85,B 0,C 180,E1 7108.603,E2 7108.603} C_VEL
LIN {X 0,Y 619.963,Z 1006.212,A -85,B 0,C 180,E1 7112.806,E2 7112.806} C_VEL
LIN {X 0,Y 619.995,Z 1001.19,A -85,B 0,C 180,E1 7116.318,E2 7116.318} C_VEL
LIN {X 0,Y 620.245,Z 989.708,A -85,B 0,C 180,E1 7120.561,E2 7120.561} C_VEL
LIN {X 0,Y 620.949,Z 973.515,A -85,B 0,C 180,E1 7124.488,E2 7124.488} C_VEL
LIN {X 0,Y 622.221,Z 952.32,A -85,B 0,C 180,E1 7128.279,E2 7128.279} C_VEL
LIN {X 0,Y 624.495,Z 924.234,A -85,B 0,C 180,E1 7132.095,E2 7132.095} C_VEL
LIN {X 0,Y 627.587,Z 889.916,A -85,B 0,C 180,E1 7135.666,E2 7135.666} C_VEL
LIN {X 0,Y 630.246,Z 858.646,A -85,B 0,C 180,E1 7138.156,E2 7138.156} C_VEL
LIN {X 0,Y 633.322,Z 819.572,A -85,B 0,C 180,E1 7140.556,E2 7140.556} C_VEL
LIN {X 0,Y 636.271,Z 776.538,A -85,B 0,C 180,E1 7142.534,E2 7142.534} C_VEL
LIN {X 0,Y 638.643,Z 731.968,A -85,B 0,C 180,E1 7143.958,E2 7143.958} C_VEL
LIN {X 0,Y 640.014,Z 687.954,A -85,B 0,C 180,E1 7144.828,E2 7144.828} C_VEL
LIN {X 0,Y 640,Z 647.519,A -85,B 0,C 180,E1 7145.372,E2 7145.372} C_VEL
LIN {X 0,Y 619.084,Z 601.31,A -85,B 0,C 180,E1 7147.155,E2 7147.155} C_VEL
LIN {X 0,Y 619.029,Z 601.31,A -85,B 0,C 180,E1 7153.269,E2 7153.269} C_VEL
LIN {X 0,Y 618.957,Z 601.31,A -85,B 0,C 180,E1 7158.635,E2 7158.635} C_VEL
LIN {X 0,Y 618.976,Z 601.31,A -85,B 0,C 180,E1 7164.027,E2 7164.027} C_VEL
LIN {X 0,Y 619.067,Z 601.31,A -85,B 0,C 180,E1 7169.075,E2 7169.075} C_VEL
LIN {X 0,Y 619.227,Z 601.31,A -85,B 0,C 180,E1 7173.872,E2 7173.872} C_VEL
LIN {X 0,Y 619.268,Z 601.31,A -85,B 0,C 180,E1 7178.471,E2 7178.471} C_VEL
LIN {X 0,Y 619.343,Z 601.31,A -85,B 0,C 180,E1 7182.93,E2 7182.93} C_VEL
LIN {X 0,Y 619.438,Z 601.31,A -85,B 0,C 180,E1 7188.716,E2 7188.716} C_VEL
LIN {X 0,Y 619.628,Z 601.31,A -85,B 0,C 180,E1 7194.386,E2 7194.386} C_VEL
LIN {X 0,Y 619.697,Z 601.31,A -85,B 0,C 180,E1 7198.597,E2 7198.597} C_VEL
LIN {X 0,Y 619.727,Z 601.31,A -85,B 0,C 180,E1 7202.8,E2 7202.8} C_VEL
LIN {X 0,Y 619.536,Z 601.31,A -85,B 0,C 180,E1 7207.021,E2 7207.021} C_VEL
LIN {X 0,Y 619.455,Z 601.31,A -85,B 0,C 180,E1 7212.713,E2 7212.713} C_VEL
LIN {X 0,Y 619.379,Z 601.31,A -85,B 0,C 180,E1 7217.42,E2 7217.42} C_VEL
LIN {X 0,Y 619.264,Z 601.31,A -85,B 0,C 180,E1 7223.04,E2 7223.04} C_VEL
LIN {X 0,Y 619.144,Z 601.31,A -85,B 0,C 180,E1 7228.227,E2 7228.227} C_VEL
LIN {X 0,Y 619.078,Z 601.31,A -85,B 0,C 180,E1 7233.672,E2 7233.672} C_VEL
LIN {X 0,Y 618.995,Z 601.31,A -85,B 0,C 180,E1 7239.514,E2 7239.514} C_VEL
LIN {X 0,Y 619.101,Z 601.31,A -85,B 0,C 180,E1 7245.2,E2 7245.2} C_VEL
LIN {X 0,Y 618.964,Z 601.31,A -85,B 0,C 180,E1 7250.466,E2 7250.466} C_VEL
LIN {X 0,Y 619.055,Z 601.31,A -85,B 0,C 180,E1 7256.302,E2 7256.302} C_VEL
LIN {X 0,Y 619.322,Z 601.31,A -85,B 0,C 180,E1 7262.152,E2 7262.152} C_VEL
LIN {X 0,Y 631.168,Z 639.21,A -85,B 0,C 180,E1 7263.39,E2 7263.39} C_VEL
LIN {X 0,Y 629.77,Z 677.898,A -85,B 0,C 180,E1 7264.599,E2 7264.599} C_VEL
LIN {X 0,Y 627.888,Z 715.151,A -85,B 0,C 180,E1 7266.318,E2 7266.318} C_VEL
LIN {X 0,Y 625.744,Z 750.403,A -85,B 0,C 180,E1 7268.605,E2 7268.605} C_VEL
LIN {X 0,Y 623.742,Z 779.963,A -85,B 0,C 180,E1 7271.2,E2 7271.2} C_VEL
LIN {X 0,Y 622.25,Z 803.615,A -85,B 0,C 180,E1 7273.943,E2 7273.943} C_VEL
LIN {X 0,Y 621.091,Z 823.136,A -85,B 0,C 180,E1 7276.954,E2 7276.954} C_VEL
LIN {X 0,Y 620.238,Z 839.524,A -85,B 0,C 180,E1 7280.505,E2 7280.505} C_VEL
LIN {X 0,Y 620.04,Z 849.546,A -85,B 0,C 180,E1 7283.683,E2 7283.683} C_VEL
LIN {X 0,Y 619.951,Z 855.923,A -85,B 0,C 180,E1 7287.194,E2 7287.194} C_VEL
LIN {X 0,Y 619.892,Z 857.39,A -85,B 0,C 180,E1 7289.996,E2 7289.996} C_VEL
LIN {X 0,Y 619.952,Z 855.818,A -85,B 0,C 180,E1 7292.798,E2 7292.798} C_VEL
LIN {X 0,Y 620.083,Z 849.333,A -85,B 0,C 180,E1 7296.309,E2 7296.309} C_VEL
LIN {X 0,Y 620.447,Z 836.481,A -85,B 0,C 180,E1 7300.194,E2 7300.194} C_VEL
LIN {X 0,Y 621.359,Z 818.496,A -85,B 0,C 180,E1 7303.75,E2 7303.75} C_VEL
LIN {X 0,Y 622.831,Z 795.703,A -85,B 0,C 180,E1 7306.97,E2 7306.97} C_VEL
LIN {X 0,Y 624.634,Z 768.06,A -85,B 0,C 180,E1 7309.849,E2 7309.849} C_VEL
LIN {X 0,Y 626.651,Z 736.614,A -85,B 0,C 180,E1 7312.287,E2 7312.287} C_VEL
LIN {X 0,Y 628.542,Z 701.756,A -85,B 0,C 180,E1 7314.284,E2 7314.284} C_VEL
LIN {X 0,Y 630.276,Z 664.43,A -85,B 0,C 180,E1 7315.799,E2 7315.799} C_VEL
LIN {X 0,Y 630.553,Z 637.012,A -85,B 0,C 180,E1 7316.602,E2 7316.602} C_VEL
LIN {X 0,Y 619.204,Z 601.31,A -85,B 0,C 180,E1 7317.772,E2 7317.772} C_VEL
LIN {X 0,Y 619.106,Z 601.31,A -85,B 0,C 180,E1 7323.705,E2 7323.705} C_VEL
LIN {X 0,Y 618.994,Z 601.31,A -85,B 0,C 180,E1 7329.522,E2 7329.522} C_VEL
LIN {X 0,Y 619.094,Z 601.31,A -85,B 0,C 180,E1 7335.21,E2 7335.21} C_VEL
LIN {X 0,Y 618.947,Z 601.31,A -85,B 0,C 180,E1 7340.482,E2 7340.482} C_VEL
LIN {X 0,Y 619.048,Z 601.31,A -85,B 0,C 180,E1 7346.318,E2 7346.318} C_VEL
LIN {X 0,Y 619.186,Z 601.31,A -85,B 0,C 180,E1 7352.302,E2 7352.302} C_VEL
LIN {X 0,Y 619.243,Z 601.31,A -85,B 0,C 180,E1 7356.959,E2 7356.959} C_VEL
LIN {X 0,Y 619.212,Z 601.31,A -85,B 0,C 180,E1 7358.936,E2 7358.936} C_VEL
LIN {X 0,Y 627.91,Z 632.571,A -85,B 0,C 180,E1 7359.69,E2 7359.69} C_VEL
LIN {X 0,Y 626.91,Z 694.876,A -85,B 0,C 180,E1 7360.608,E2 7360.608} C_VEL
LIN {X 0,Y 625.912,Z 730.634,A -85,B 0,C 180,E1 7361.709,E2 7361.709} C_VEL
LIN {X 0,Y 624.514,Z 763.035,A -85,B 0,C 180,E1 7363.28,E2 7363.28} C_VEL
LIN {X 0,Y 623.207,Z 792.056,A -85,B 0,C 180,E1 7365.304,E2 7365.304} C_VEL
LIN {X 0,Y 622.044,Z 816.801,A -85,B 0,C 180,E1 7367.698,E2 7367.698} C_VEL
LIN {X 0,Y 621.221,Z 837.589,A -85,B 0,C 180,E1 7370.532,E2 7370.532} C_VEL
LIN {X 0,Y 620.77,Z 851.626,A -85,B 0,C 180,E1 7373.345,E2 7373.345} C_VEL
LIN {X 0,Y 620.562,Z 861.199,A -85,B 0,C 180,E1 7376.503,E2 7376.503} C_VEL
LIN {X 0,Y 620.484,Z 864.282,A -85,B 0,C 180,E1 7378.603,E2 7378.603} C_VEL
LIN {X 0,Y 620.524,Z 864.572,A -85,B 0,C 180,E1 7381.401,E2 7381.401} C_VEL
LIN {X 0,Y 620.715,Z 860.418,A -85,B 0,C 180,E1 7384.201,E2 7384.201} C_VEL
LIN {X 0,Y 621.074,Z 851.454,A -85,B 0,C 180,E1 7387.007,E2 7387.007} C_VEL
LIN {X 0,Y 621.719,Z 835.862,A -85,B 0,C 180,E1 7389.999,E2 7389.999} C_VEL
LIN {X 0,Y 622.588,Z 815.35,A -85,B 0,C 180,E1 7392.651,E2 7392.651} C_VEL
LIN {X 0,Y 623.834,Z 790.388,A -85,B 0,C 180,E1 7394.954,E2 7394.954} C_VEL
LIN {X 0,Y 625.061,Z 760.772,A -85,B 0,C 180,E1 7396.909,E2 7396.909} C_VEL
LIN {X 0,Y 626.329,Z 726.563,A -85,B 0,C 180,E1 7398.465,E2 7398.465} C_VEL
LIN {X 0,Y 627.483,Z 689.444,A -85,B 0,C 180,E1 7399.526,E2 7399.526} C_VEL
LIN {X 0,Y 628.191,Z 627.771,A -85,B 0,C 180,E1 7400.527,E2 7400.527} C_VEL
LIN {X 0,Y 619.268,Z 601.31,A -85,B 0,C 180,E1 7401.455,E2 7401.455} C_VEL
LIN {X 0,Y 619.176,Z 601.31,A -85,B 0,C 180,E1 7406.131,E2 7406.131} C_VEL
LIN {X 0,Y 619.091,Z 601.31,A -85,B 0,C 180,E1 7411.069,E2 7411.069} C_VEL
LIN {X 0,Y 619.057,Z 601.31,A -85,B 0,C 180,E1 7412.243,E2 7412.243} C_VEL
LIN {X 0,Y 616.583,Z 601.31,A -85,B 0,C 180,E1 7413.429,E2 7413.429} C_VEL
LIN {X 0,Y 611.187,Z 601.31,A -85,B 0,C 180,E1 7415.202,E2 7415.202} C_VEL
LIN {X 0,Y 611.08,Z 601.31,A -85,B 0,C 180,E1 7415.407,E2 7415.407} C_VEL
LIN {X 0,Y 611.115,Z 601.31,A -85,B 0,C 180,E1 7420.131,E2 7420.131} C_VEL
LIN {X 0,Y 611.074,Z 601.31,A -85,B 0,C 180,E1 7426.035,E2 7426.035} C_VEL
LIN {X 0,Y 611.003,Z 601.31,A -85,B 0,C 180,E1 7431.691,E2 7431.691} C_VEL
LIN {X 0,Y 611.137,Z 601.419,A -85,B 0,C 180,E1 7433.17,E2 7433.17} C_VEL
LIN {X 0,Y 625.84,Z 640.158,A -85,B 0,C 180,E1 7434.318,E2 7434.318} C_VEL
LIN {X 0,Y 631.686,Z 652.58,A -85,B 0,C 180,E1 7434.709,E2 7434.709} C_VEL
LIN {X 0,Y 630.997,Z 712.872,A -85,B 0,C 180,E1 7435.538,E2 7435.538} C_VEL
LIN {X 0,Y 629.097,Z 759.007,A -85,B 0,C 180,E1 7436.734,E2 7436.734} C_VEL
LIN {X 0,Y 626.633,Z 803.134,A -85,B 0,C 180,E1 7438.478,E2 7438.478} C_VEL
LIN {X 0,Y 623.844,Z 843.158,A -85,B 0,C 180,E1 7440.643,E2 7440.643} C_VEL
LIN {X 0,Y 620.922,Z 880.075,A -85,B 0,C 180,E1 7443.241,E2 7443.241} C_VEL
LIN {X 0,Y 618.456,Z 907.761,A -85,B 0,C 180,E1 7445.776,E2 7445.776} C_VEL
LIN {X 0,Y 615.742,Z 936.754,A -85,B 0,C 180,E1 7449.216,E2 7449.216} C_VEL
LIN {X 0,Y 613.781,Z 962.288,A -85,B 0,C 180,E1 7453.142,E2 7453.142} C_VEL
LIN {X 0,Y 612.697,Z 981.624,A -85,B 0,C 180,E1 7457.144,E2 7457.144} C_VEL
LIN {X 0,Y 612.257,Z 994.245,A -85,B 0,C 180,E1 7460.747,E2 7460.747} C_VEL
LIN {X 0,Y 612.104,Z 1003.673,A -85,B 0,C 180,E1 7465.034,E2 7465.034} C_VEL
LIN {X 0,Y 612.062,Z 1007.167,A -85,B 0,C 180,E1 7468.585,E2 7468.585} C_VEL
LIN {X 0,Y 612.056,Z 1006.211,A -85,B 0,C 180,E1 7472.842,E2 7472.842} C_VEL
LIN {X 0,Y 612.093,Z 1001.19,A -85,B 0,C 180,E1 7476.4,E2 7476.4} C_VEL
LIN {X 0,Y 612.377,Z 989.708,A -85,B 0,C 180,E1 7480.698,E2 7480.698} C_VEL
LIN {X 0,Y 613.14,Z 973.674,A -85,B 0,C 180,E1 7484.643,E2 7484.643} C_VEL
LIN {X 0,Y 614.502,Z 952.319,A -85,B 0,C 180,E1 7488.517,E2 7488.517} C_VEL
LIN {X 0,Y 616.924,Z 924.373,A -85,B 0,C 180,E1 7492.364,E2 7492.364} C_VEL
LIN {X 0,Y 619.889,Z 892.779,A -85,B 0,C 180,E1 7495.694,E2 7495.694} C_VEL
LIN {X 0,Y 622.949,Z 856.748,A -85,B 0,C 180,E1 7498.547,E2 7498.547} C_VEL
LIN {X 0,Y 626.102,Z 817.75,A -85,B 0,C 180,E1 7500.946,E2 7500.946} C_VEL
LIN {X 0,Y 629.249,Z 774.427,A -85,B 0,C 180,E1 7502.933,E2 7502.933} C_VEL
LIN {X 0,Y 631.738,Z 729.209,A -85,B 0,C 180,E1 7504.372,E2 7504.372} C_VEL
LIN {X 0,Y 633.231,Z 682.421,A -85,B 0,C 180,E1 7505.254,E2 7505.254} C_VEL
LIN {X 0,Y 633.095,Z 650.059,A -85,B 0,C 180,E1 7505.695,E2 7505.695} C_VEL
LIN {X 0,Y 611.128,Z 601.31,A -85,B 0,C 180,E1 7507.618,E2 7507.618} C_VEL
LIN {X 0,Y 611.078,Z 601.31,A -85,B 0,C 180,E1 7512.032,E2 7512.032} C_VEL
LIN {X 0,Y 611.034,Z 601.31,A -85,B 0,C 180,E1 7518.072,E2 7518.072} C_VEL
LIN {X 0,Y 611.025,Z 601.31,A -85,B 0,C 180,E1 7523.484,E2 7523.484} C_VEL
LIN {X 0,Y 611.128,Z 601.31,A -85,B 0,C 180,E1 7528.628,E2 7528.628} C_VEL
LIN {X 0,Y 611.277,Z 601.31,A -85,B 0,C 180,E1 7533.506,E2 7533.506} C_VEL
LIN {X 0,Y 611.375,Z 601.31,A -85,B 0,C 180,E1 7538.179,E2 7538.179} C_VEL
LIN {X 0,Y 611.438,Z 601.31,A -85,B 0,C 180,E1 7542.702,E2 7542.702} C_VEL
LIN {X 0,Y 611.547,Z 601.31,A -85,B 0,C 180,E1 7548.568,E2 7548.568} C_VEL
LIN {X 0,Y 611.719,Z 601.31,A -85,B 0,C 180,E1 7554.313,E2 7554.313} C_VEL
LIN {X 0,Y 611.796,Z 601.31,A -85,B 0,C 180,E1 7558.579,E2 7558.579} C_VEL
LIN {X 0,Y 611.823,Z 601.31,A -85,B 0,C 180,E1 7562.837,E2 7562.837} C_VEL
LIN {X 0,Y 611.593,Z 601.31,A -85,B 0,C 180,E1 7567.668,E2 7567.668} C_VEL
LIN {X 0,Y 611.534,Z 601.31,A -85,B 0,C 180,E1 7572.88,E2 7572.88} C_VEL
LIN {X 0,Y 611.491,Z 601.31,A -85,B 0,C 180,E1 7577.293,E2 7577.293} C_VEL
LIN {X 0,Y 611.386,Z 601.31,A -85,B 0,C 180,E1 7581.817,E2 7581.817} C_VEL
LIN {X 0,Y 611.254,Z 601.31,A -85,B 0,C 180,E1 7586.817,E2 7586.817} C_VEL
LIN {X 0,Y 611.165,Z 601.31,A -85,B 0,C 180,E1 7592.542,E2 7592.542} C_VEL
LIN {X 0,Y 611.079,Z 601.31,A -85,B 0,C 180,E1 7598.296,E2 7598.296} C_VEL
LIN {X 0,Y 611.139,Z 601.31,A -85,B 0,C 180,E1 7604.022,E2 7604.022} C_VEL
LIN {X 0,Y 611.069,Z 601.31,A -85,B 0,C 180,E1 7610.218,E2 7610.218} C_VEL
LIN {X 0,Y 611.059,Z 601.31,A -85,B 0,C 180,E1 7615.223,E2 7615.223} C_VEL
LIN {X 0,Y 611.199,Z 601.31,A -85,B 0,C 180,E1 7620.272,E2 7620.272} C_VEL
LIN {X 0,Y 611.395,Z 601.31,A -85,B 0,C 180,E1 7621.799,E2 7621.799} C_VEL
LIN {X 0,Y 623.74,Z 642.653,A -85,B 0,C 180,E1 7623.213,E2 7623.213} C_VEL
LIN {X 0,Y 622.067,Z 682.817,A -85,B 0,C 180,E1 7624.536,E2 7624.536} C_VEL
LIN {X 0,Y 620.023,Z 721.101,A -85,B 0,C 180,E1 7626.415,E2 7626.415} C_VEL
LIN {X 0,Y 617.976,Z 753.064,A -85,B 0,C 180,E1 7628.566,E2 7628.566} C_VEL
LIN {X 0,Y 616.049,Z 781.231,A -85,B 0,C 180,E1 7631.082,E2 7631.082} C_VEL
LIN {X 0,Y 614.399,Z 806.357,A -85,B 0,C 180,E1 7634.063,E2 7634.063} C_VEL
LIN {X 0,Y 613.242,Z 825.701,A -85,B 0,C 180,E1 7637.148,E2 7637.148} C_VEL
LIN {X 0,Y 612.476,Z 840.372,A -85,B 0,C 180,E1 7640.383,E2 7640.383} C_VEL
LIN {X 0,Y 612.207,Z 850.183,A -85,B 0,C 180,E1 7643.602,E2 7643.602} C_VEL
LIN {X 0,Y 612.056,Z 856.241,A -85,B 0,C 180,E1 7647.158,E2 7647.158} C_VEL
LIN {X 0,Y 611.997,Z 857.649,A -85,B 0,C 180,E1 7649.996,E2 7649.996} C_VEL
LIN {X 0,Y 612.058,Z 856.145,A -85,B 0,C 180,E1 7652.834,E2 7652.834} C_VEL
LIN {X 0,Y 612.248,Z 849.981,A -85,B 0,C 180,E1 7656.39,E2 7656.39} C_VEL
LIN {X 0,Y 612.597,Z 838.703,A -85,B 0,C 180,E1 7659.966,E2 7659.966} C_VEL
LIN {X 0,Y 613.436,Z 822.274,A -85,B 0,C 180,E1 7663.385,E2 7663.385} C_VEL
LIN {X 0,Y 614.837,Z 800.199,A -85,B 0,C 180,E1 7666.659,E2 7666.659} C_VEL
LIN {X 0,Y 616.652,Z 773.829,A -85,B 0,C 180,E1 7669.555,E2 7669.555} C_VEL
LIN {X 0,Y 618.603,Z 743.897,A -85,B 0,C 180,E1 7672.024,E2 7672.024} C_VEL
LIN {X 0,Y 620.76,Z 708.963,A -85,B 0,C 180,E1 7674.165,E2 7674.165} C_VEL
LIN {X 0,Y 622.671,Z 670.077,A -85,B 0,C 180,E1 7675.858,E2 7675.858} C_VEL
LIN {X 0,Y 623.114,Z 638.842,A -85,B 0,C 180,E1 7676.825,E2 7676.825} C_VEL
LIN {X 0,Y 611.3,Z 601.31,A -85,B 0,C 180,E1 7678.155,E2 7678.155} C_VEL
LIN {X 0,Y 611.19,Z 601.31,A -85,B 0,C 180,E1 7683.048,E2 7683.048} C_VEL
LIN {X 0,Y 611.069,Z 601.31,A -85,B 0,C 180,E1 7688.304,E2 7688.304} C_VEL
LIN {X 0,Y 611.151,Z 601.31,A -85,B 0,C 180,E1 7694.044,E2 7694.044} C_VEL
LIN {X 0,Y 611.05,Z 601.31,A -85,B 0,C 180,E1 7700.231,E2 7700.231} C_VEL
LIN {X 0,Y 611.056,Z 601.31,A -85,B 0,C 180,E1 7705.238,E2 7705.238} C_VEL
LIN {X 0,Y 611.188,Z 601.31,A -85,B 0,C 180,E1 7710.285,E2 7710.285} C_VEL
LIN {X 0,Y 611.327,Z 601.31,A -85,B 0,C 180,E1 7715.088,E2 7715.088} C_VEL
LIN {X 0,Y 611.308,Z 601.31,A -85,B 0,C 180,E1 7718.64,E2 7718.64} C_VEL
LIN {X 0,Y 620.551,Z 633.451,A -85,B 0,C 180,E1 7719.439,E2 7719.439} C_VEL
LIN {X 0,Y 619.475,Z 694.984,A -85,B 0,C 180,E1 7720.365,E2 7720.365} C_VEL
LIN {X 0,Y 618.419,Z 730.775,A -85,B 0,C 180,E1 7721.479,E2 7721.479} C_VEL
LIN {X 0,Y 616.907,Z 764.242,A -85,B 0,C 180,E1 7723.123,E2 7723.123} C_VEL
LIN {X 0,Y 615.521,Z 793.543,A -85,B 0,C 180,E1 7725.208,E2 7725.208} C_VEL
LIN {X 0,Y 614.26,Z 818.873,A -85,B 0,C 180,E1 7727.721,E2 7727.721} C_VEL
LIN {X 0,Y 613.451,Z 838.389,A -85,B 0,C 180,E1 7730.427,E2 7730.427} C_VEL
LIN {X 0,Y 612.981,Z 852.454,A -85,B 0,C 180,E1 7733.26,E2 7733.26} C_VEL
LIN {X 0,Y 612.728,Z 862.14,A -85,B 0,C 180,E1 7736.458,E2 7736.458} C_VEL
LIN {X 0,Y 612.662,Z 865.282,A -85,B 0,C 180,E1 7738.585,E2 7738.585} C_VEL
LIN {X 0,Y 612.703,Z 865.626,A -85,B 0,C 180,E1 7741.419,E2 7741.419} C_VEL
LIN {X 0,Y 612.905,Z 861.49,A -85,B 0,C 180,E1 7744.254,E2 7744.254} C_VEL
LIN {X 0,Y 613.322,Z 852.53,A -85,B 0,C 180,E1 7747.096,E2 7747.096} C_VEL
LIN {X 0,Y 614.01,Z 836.899,A -85,B 0,C 180,E1 7750.126,E2 7750.126} C_VEL
LIN {X 0,Y 614.92,Z 816.319,A -85,B 0,C 180,E1 7752.812,E2 7752.812} C_VEL
LIN {X 0,Y 616.26,Z 791.324,A -85,B 0,C 180,E1 7755.142,E2 7755.142} C_VEL
